Omron Sysmac Studio project 20-1203_20210423 (Sysmac Studio 1.44.0.15, StandardProject)

# Controller new_Controller_0: NX1P2-1140DT version 1.42
Units and slaves: 節點1 : ASDA-A2-E CoE Drive (E001); 節點2 : ASDA-A2-E CoE Drive (E002); 節點3 : ASDA-A2-E CoE Drive (E003); 節點4 : ASDA-A2-E CoE Drive (E004)
Axis MC_AxisLSt5, settings changed from default: AxisType=ServoType, UnitsConversion=EnumElement5, UnitsNumerator=1280000, UnitsDenominator=120, TravelDistancePerWorkRotation=360, WorkGearRatio=3, MaxVelocity=18000, MaxJogVelocity=1800, InPositionCheckTime=500, ZeroPositionBand=0.05
Axis MC_AxisRSt5, settings changed from default: AxisNumber=1, AxisType=ServoType, UnitsConversion=EnumElement5, UnitsNumerator=1280000, UnitsDenominator=120, TravelDistancePerWorkRotation=360, WorkGearRatio=3, MaxVelocity=18000, MaxJogVelocity=1800, InPositionCheckTime=500, ZeroPositionBand=0.05
Axis MC_AxisLSt6, settings changed from default: AxisNumber=2, AxisType=ServoType, UnitsConversion=EnumElement5, UnitsNumerator=1280000, UnitsDenominator=120, TravelDistancePerWorkRotation=360, WorkGearRatio=3, MaxVelocity=18000, MaxJogVelocity=1800, InPositionCheckTime=500, ZeroPositionBand=0.05
Axis MC_AxisRSt6, settings changed from default: AxisNumber=3, AxisType=ServoType, UnitsConversion=EnumElement5, UnitsNumerator=1280000, UnitsDenominator=120, TravelDistancePerWorkRotation=360, WorkGearRatio=3, MaxVelocity=18000, MaxJogVelocity=1800, InPositionCheckTime=500, ZeroPositionBand=0.05
Task PrimaryTask (priority 4, period or condition 4000): prAxisDefineSt5L, prAxisDefineSt5R, prAxisDefineSt6L, prAxisDefineSt6R, prInitial, prIndex, prBowlFeeder, prError, prStation2, prStation3, prStation7, prStation8, prStart, prFeedScrewS5, prCommProgram, prFeedScrewS6, prCycleTime, prBZAndLight, prStation5, prStation6

TYPE StationRecord : STRUCT
    FinishFlag : ARRAY[0..19] OF BOOL;
    OKFlag_1 : ARRAY[0..19] OF BOOL;
    OKFlag_2 : ARRAY[0..19] OF BOOL;
    OKFlag_3 : ARRAY[0..19] OF BOOL;
    OKFlag_4 : ARRAY[0..19] OF BOOL;
    NGFlag_1 : ARRAY[0..19] OF BOOL;
    NGFlag_2 : ARRAY[0..19] OF BOOL;
    NGFlag_3 : ARRAY[0..19] OF BOOL;
    NGFlag_4 : ARRAY[0..19] OF BOOL;
    ErrorRecordData : ARRAY[0..19] OF INT;
END_STRUCT END_TYPE

VAR_GLOBAL CONSTANT
    MC_AxisLSt5 : _sAXIS_REF;  (* at MC://_MC_AX[0] *)
    MC_AxisRSt5 : _sAXIS_REF;  (* at MC://_MC_AX[1] *)
    MC_AxisLSt6 : _sAXIS_REF;  (* at MC://_MC_AX[2] *)
    MC_AxisRSt6 : _sAXIS_REF;  (* at MC://_MC_AX[3] *)
END_VAR
VAR_GLOBAL
    PB_Start1 : BOOL;  (* in_input; at BuiltInIO://cpu/#0/Input_Bit_00; published *)
    PB_Reset1 : BOOL;  (* in_input; at BuiltInIO://cpu/#0/Input_Bit_01; published *)
    PB_Estop1 : BOOL;  (* in_input; at BuiltInIO://cpu/#0/Input_Bit_02; published *)
    PB_Start2 : BOOL;  (* in_input; at BuiltInIO://cpu/#0/Input_Bit_03; published *)
    PB_Reset2 : BOOL;  (* in_input; at BuiltInIO://cpu/#0/Input_Bit_04; published *)
    PB_Estop2 : BOOL;  (* in_input; at BuiltInIO://cpu/#0/Input_Bit_05; published *)
    SNR_AirSource : BOOL;  (* in_input; at BuiltInIO://cpu/#0/Input_Bit_06; published *)
    SNR_Index : BOOL;  (* in_input; at BuiltInIO://cpu/#0/Input_Bit_07; published *)
    LS_S2_THBack1 : BOOL;  (* in_input; at BuiltInIO://cpu/#0/Input_Bit_08; published *)
    LS_S2_THOut1 : BOOL;  (* in_input; at BuiltInIO://cpu/#0/Input_Bit_09; published *)
    LS_S2_THBack2 : BOOL;  (* in_input; at BuiltInIO://cpu/#0/Input_Bit_10; published *)
    LS_S2_THOut2 : BOOL;  (* in_input; at BuiltInIO://cpu/#0/Input_Bit_11; published *)
    LS_S2_MoveBack : BOOL;  (* in_input; at BuiltInIO://cpu/#0/Input_Bit_12; published *)
    LS_S2_MoveOut : BOOL;  (* in_input; at BuiltInIO://cpu/#0/Input_Bit_13; published *)
    SNR_S2_Feed : BOOL;  (* in_input; at BuiltInIO://cpu/#0/Input_Bit_14; published *)
    SNR_S2_Full : BOOL;  (* in_input; at BuiltInIO://cpu/#0/Input_Bit_15; published *)
    LS_S3_THBack1 : BOOL;  (* in_input; at BuiltInIO://cpu/#0/Input_Bit_16; published *)
    LS_S3_THOut1 : BOOL;  (* in_input; at BuiltInIO://cpu/#0/Input_Bit_17; published *)
    LS_S3_THBack2 : BOOL;  (* in_input; at BuiltInIO://cpu/#0/Input_Bit_18; published *)
    LS_S3_THOut2 : BOOL;  (* in_input; at BuiltInIO://cpu/#0/Input_Bit_19; published *)
    LS_S3_MoveBack : BOOL;  (* in_input; at BuiltInIO://cpu/#0/Input_Bit_20; published *)
    LS_S3_MoveOut : BOOL;  (* in_input; at BuiltInIO://cpu/#0/Input_Bit_21; published *)
    SNR_S3_Feed : BOOL;  (* in_input; at BuiltInIO://cpu/#0/Input_Bit_22; published *)
    SNR_S3_Full : BOOL;  (* in_input; at BuiltInIO://cpu/#0/Input_Bit_23; published *)
    LS_S5_UpDownBack : BOOL;  (* in_input; at IOBus://unit#2/Input Bit 16 bits/Input Bit 00; published *)
    LS_S5_UpDownOut : BOOL;  (* in_input; at IOBus://unit#2/Input Bit 16 bits/Input Bit 01; published *)
    LS_S5_FixBack : BOOL;  (* in_input; at IOBus://unit#2/Input Bit 16 bits/Input Bit 02; published *)
    LS_S5_FixOut : BOOL;  (* in_input; at IOBus://unit#2/Input Bit 16 bits/Input Bit 03; published *)
    SNR_S5_L_Check : BOOL;  (* in_input; at IOBus://unit#2/Input Bit 16 bits/Input Bit 04; published *)
    SNR_S5_R_Check : BOOL;  (* in_input; at IOBus://unit#2/Input Bit 16 bits/Input Bit 05; published *)
    SNR_S5_L_Feed : BOOL;  (* in_input; at IOBus://unit#2/Input Bit 16 bits/Input Bit 06; published *)
    SNR_S5_R_Feed : BOOL;  (* in_input; at IOBus://unit#2/Input Bit 16 bits/Input Bit 07; published *)
    LS_S6_UpDownBack : BOOL;  (* in_input; at IOBus://unit#2/Input Bit 16 bits/Input Bit 08; published *)
    LS_S6_UpDownOut : BOOL;  (* in_input; at IOBus://unit#2/Input Bit 16 bits/Input Bit 09; published *)
    LS_S6_FixBack : BOOL;  (* in_input; at IOBus://unit#2/Input Bit 16 bits/Input Bit 10; published *)
    LS_S6_FixOut : BOOL;  (* in_input; at IOBus://unit#2/Input Bit 16 bits/Input Bit 11; published *)
    SNR_S6_L_Check : BOOL;  (* in_input; at IOBus://unit#2/Input Bit 16 bits/Input Bit 12; published *)
    SNR_S6_R_Check : BOOL;  (* in_input; at IOBus://unit#2/Input Bit 16 bits/Input Bit 13; published *)
    SNR_S6_L_Feed : BOOL;  (* in_input; at IOBus://unit#2/Input Bit 16 bits/Input Bit 14; published *)
    SNR_S6_R_Feed : BOOL;  (* in_input; at IOBus://unit#2/Input Bit 16 bits/Input Bit 15; published *)
    SNR_S5_Full : BOOL;  (* in_input; at IOBus://unit#3/Input Bit 16 bits/Input Bit 00; published *)
    SNR_S6_Full : BOOL;  (* in_input; at IOBus://unit#3/Input Bit 16 bits/Input Bit 01; published *)
    LS_S7_MoveBack1 : BOOL;  (* in_input; at IOBus://unit#3/Input Bit 16 bits/Input Bit 02; published *)
    LS_S7_MoveOut1 : BOOL;  (* in_input; at IOBus://unit#3/Input Bit 16 bits/Input Bit 03; published *)
    LS_S7_MoveBack2 : BOOL;  (* in_input; at IOBus://unit#3/Input Bit 16 bits/Input Bit 04; published *)
    LS_S7_MoveOut2 : BOOL;  (* in_input; at IOBus://unit#3/Input Bit 16 bits/Input Bit 05; published *)
    LS_S7_MoveBack3 : BOOL;  (* in_input; at IOBus://unit#3/Input Bit 16 bits/Input Bit 06; published *)
    LS_S7_MoveOut3 : BOOL;  (* in_input; at IOBus://unit#3/Input Bit 16 bits/Input Bit 07; published *)
    LS_S7_MoveBack4 : BOOL;  (* in_input; at IOBus://unit#3/Input Bit 16 bits/Input Bit 08; published *)
    LS_S7_MoveOut4 : BOOL;  (* in_input; at IOBus://unit#3/Input Bit 16 bits/Input Bit 09; published *)
    SNR_S7_Full : BOOL;  (* in_input; at IOBus://unit#3/Input Bit 16 bits/Input Bit 10; published *)
    LS_S8_MoveBack : BOOL;  (* in_input; at IOBus://unit#3/Input Bit 16 bits/Input Bit 11; published *)
    LS_S8_MoveOut : BOOL;  (* in_input; at IOBus://unit#3/Input Bit 16 bits/Input Bit 12; published *)
    LS_S5_IndexFixBack : BOOL;  (* in_input; at IOBus://unit#3/Input Bit 16 bits/Input Bit 13; published *)
    LS_S5_IndexFixOut : BOOL;  (* in_input; at IOBus://unit#3/Input Bit 16 bits/Input Bit 14; published *)
    LS_S6_IndexFixBack : BOOL;  (* in_input; at IOBus://unit#3/Input Bit 16 bits/Input Bit 15; published *)
    LS_S6_IndexFixOut : BOOL;  (* in_input; at IOBus://unit#4/Input Bit 16 bits/Input Bit 00; published *)
    RY_Index : BOOL;  (* output; at BuiltInIO://cpu/#0/Output_Bit_00; published *)
    RY_S2_Full : BOOL;  (* output; at BuiltInIO://cpu/#0/Output_Bit_01; published *)
    RY_S2_Feed : BOOL;  (* output; at BuiltInIO://cpu/#0/Output_Bit_02; published *)
    RY_S3_Full : BOOL;  (* output; at BuiltInIO://cpu/#0/Output_Bit_03; published *)
    RY_S3_Feed : BOOL;  (* output; at BuiltInIO://cpu/#0/Output_Bit_04; published *)
    RY_S5_Full : BOOL;  (* output; at BuiltInIO://cpu/#0/Output_Bit_05; published *)
    RY_S5_Feed : BOOL;  (* output; at BuiltInIO://cpu/#0/Output_Bit_06; published *)
    RY_S6_Full : BOOL;  (* output; at BuiltInIO://cpu/#0/Output_Bit_07; published *)
    RY_S6_Feed : BOOL;  (* output; at BuiltInIO://cpu/#0/Output_Bit_08; published *)
    SOL_S2_THBack1 : BOOL;  (* output; at BuiltInIO://cpu/#0/Output_Bit_09; published *)
    SOL_S2_THOut1 : BOOL;  (* output; at BuiltInIO://cpu/#0/Output_Bit_10; published *)
    SOL_S2_THBack2 : BOOL;  (* output; at BuiltInIO://cpu/#0/Output_Bit_11; published *)
    SOL_S2_THOut2 : BOOL;  (* output; at BuiltInIO://cpu/#0/Output_Bit_12; published *)
    SOL_S2_Move : BOOL;  (* output; at BuiltInIO://cpu/#0/Output_Bit_13; published *)
    SOL_S3_THBack1 : BOOL;  (* output; at BuiltInIO://cpu/#0/Output_Bit_14; published *)
    SOL_S3_THOut1 : BOOL;  (* output; at BuiltInIO://cpu/#0/Output_Bit_15; published *)
    SOL_S3_THBack2 : BOOL;  (* output; at IOBus://unit#5/Output Bit 16 bits/Output Bit 00; published *)
    SOL_S3_THOut2 : BOOL;  (* output; at IOBus://unit#5/Output Bit 16 bits/Output Bit 01; published *)
    SOL_S3_Move : BOOL;  (* output; at IOBus://unit#5/Output Bit 16 bits/Output Bit 02; published *)
    SOL_S5_Feed : BOOL;  (* output; at IOBus://unit#5/Output Bit 16 bits/Output Bit 03; published *)
    SOL_S5_UpDown : BOOL;  (* output; at IOBus://unit#5/Output Bit 16 bits/Output Bit 04; published *)
    SOL_S5_Clamp : BOOL;  (* output; at IOBus://unit#5/Output Bit 16 bits/Output Bit 05; published *)
    SOL_S5_Fix : BOOL;  (* output; at IOBus://unit#5/Output Bit 16 bits/Output Bit 06; published *)
    SOL_S6_Feed : BOOL;  (* output; at IOBus://unit#5/Output Bit 16 bits/Output Bit 07; published *)
    SOL_S6_UpDown : BOOL;  (* output; at IOBus://unit#5/Output Bit 16 bits/Output Bit 08; published *)
    SOL_S6_Clamp : BOOL;  (* output; at IOBus://unit#5/Output Bit 16 bits/Output Bit 09; published *)
    SOL_S6_Fix : BOOL;  (* output; at IOBus://unit#5/Output Bit 16 bits/Output Bit 10; published *)
    SOL_S7_Move1 : BOOL;  (* output; at IOBus://unit#5/Output Bit 16 bits/Output Bit 11; published *)
    SOL_S7_Move2 : BOOL;  (* output; at IOBus://unit#5/Output Bit 16 bits/Output Bit 12; published *)
    SOL_S7_Move3 : BOOL;  (* output; at IOBus://unit#5/Output Bit 16 bits/Output Bit 13; published *)
    SOL_S7_Move4 : BOOL;  (* output; at IOBus://unit#5/Output Bit 16 bits/Output Bit 14; published *)
    SOL_S8_Move : BOOL;  (* output; at IOBus://unit#5/Output Bit 16 bits/Output Bit 15; published *)
    SOL_S5_IndexFixBack : BOOL;  (* output; at IOBus://unit#6/Output Bit 16 bits/Output Bit 00; published *)
    SOL_S5_IndexFixOut : BOOL;  (* output; at IOBus://unit#6/Output Bit 16 bits/Output Bit 01; published *)
    SOL_S6_IndexFixBack : BOOL;  (* output; at IOBus://unit#6/Output Bit 16 bits/Output Bit 02; published *)
    SOL_S6_IndexFixOut : BOOL;  (* output; at IOBus://unit#6/Output Bit 16 bits/Output Bit 03; published *)
    BZ : BOOL;  (* output; at IOBus://unit#6/Output Bit 16 bits/Output Bit 04; published *)
    YL : BOOL;  (* output; at IOBus://unit#6/Output Bit 16 bits/Output Bit 05; published *)
    GL : BOOL;  (* output; at IOBus://unit#6/Output Bit 16 bits/Output Bit 06; published *)
    RL : BOOL;  (* output; at IOBus://unit#6/Output Bit 16 bits/Output Bit 07; published *)
    SOL_S2_Fix : BOOL;  (* output; at IOBus://unit#6/Output Bit 16 bits/Output Bit 08; published *)
    SOL_S3_Fix : BOOL;  (* output; at IOBus://unit#6/Output Bit 16 bits/Output Bit 09; published *)
END_VAR
VAR_GLOBAL RETAIN
    HMI_FeedScrewTime : ARRAY[0..1] OF INT;  (* published *)
END_VAR
VAR_GLOBAL
    HMIPB_RY_Index : BOOL;  (* HMIPB; published *)
    HMIPB_SOL_S2_THBack1 : BOOL;  (* HMIPB; published *)
    HMIPB_SOL_S2_THOut1 : BOOL;  (* HMIPB; published *)
    HMIPB_SOL_S2_THBack2 : BOOL;  (* HMIPB; published *)
    HMIPB_SOL_S2_THOut2 : BOOL;  (* HMIPB; published *)
    HMIPB_SOL_S2_Move : BOOL;  (* HMIPB; published *)
    HMIPB_SOL_S3_THBack1 : BOOL;  (* HMIPB; published *)
    HMIPB_SOL_S3_THOut1 : BOOL;  (* HMIPB; published *)
    HMIPB_SOL_S3_THBack2 : BOOL;  (* HMIPB; published *)
    HMIPB_SOL_S3_THOut2 : BOOL;  (* HMIPB; published *)
    HMIPB_SOL_S3_Move : BOOL;  (* HMIPB; published *)
    HMIPB_SOL_S5_Feed : BOOL;  (* HMIPB; published *)
    HMIPB_SOL_S5_UpDown : BOOL;  (* HMIPB; published *)
    HMIPB_SOL_S5_Clamp : BOOL;  (* HMIPB; published *)
    HMIPB_SOL_S5_Fix : BOOL;  (* HMIPB; published *)
    HMIPB_SOL_S6_Feed : BOOL;  (* HMIPB; published *)
    HMIPB_SOL_S6_UpDown : BOOL;  (* HMIPB; published *)
    HMIPB_SOL_S6_Clamp : BOOL;  (* HMIPB; published *)
    HMIPB_SOL_S6_Fix : BOOL;  (* HMIPB; published *)
    HMIPB_SOL_S7_Move1 : BOOL;  (* HMIPB; published *)
    HMIPB_SOL_S7_Move2 : BOOL;  (* HMIPB; published *)
    HMIPB_SOL_S7_Move3 : BOOL;  (* HMIPB; published *)
    HMIPB_SOL_S7_Move4 : BOOL;  (* HMIPB; published *)
    HMIPB_SOL_S8_Move : BOOL;  (* HMIPB; published *)
    HMIPB_SOL_IndexFixBack : BOOL;  (* HMIPB; published *)
    HMIPB_SOL_IndexFixOut : BOOL;  (* HMIPB; published *)
    HMIPB_SOL_S2_Fix : BOOL;  (* HMIPB; published *)
    HMIPB_SOL_S3_Fix : BOOL;  (* HMIPB; published *)
    HMIPB_S2Feed : BOOL;  (* published *)
    HMIPB_S3Feed : BOOL;  (* published *)
    HMIPB_S5Feed : BOOL;  (* published *)
    HMIPB_S6Feed : BOOL;  (* published *)
    HMIPB_DisableS2 : BOOL;  (* published *)
    HMIPB_DisableS3 : BOOL;  (* published *)
    BackoutStart : ARRAY[0..3] OF BOOL;
    BackoutBusy : ARRAY[0..3] OF BOOL;
    ScrewStartS5LFW : BOOL;
    ScrewStartS5LRW : BOOL;
    ScrewStartS5RFW : BOOL;
    ScrewStartS5RRW : BOOL;
    ScrewStartS6LFW : BOOL;
    ScrewStartS6LRW : BOOL;
    ScrewStartS6RFW : BOOL;
    ScrewStartS6RRW : BOOL;
    Error_PB_Estop1 : BOOL;  (* Error; published *)
    Error_PB_Estop2 : BOOL;  (* Error; published *)
    Error_SNR_AirSource : BOOL;  (* Error; published *)
    Error_SNR_Index : BOOL;  (* Error; published *)
    Error_LS_S2_THBack1 : BOOL;  (* Error; published *)
    Error_LS_S2_THOut1 : BOOL;  (* Error; published *)
    Error_LS_S2_THBack2 : BOOL;  (* Error; published *)
    Error_LS_S2_THOut2 : BOOL;  (* Error; published *)
    Error_LS_S2_MoveBack : BOOL;  (* Error; published *)
    Error_LS_S2_MoveOut : BOOL;  (* Error; published *)
    Error_SNR_S2_Feed : BOOL;  (* Error; published *)
    Error_SNR_S2_Full : BOOL;  (* Error; published *)
    Error_LS_S3_THBack1 : BOOL;  (* Error; published *)
    Error_LS_S3_THOut1 : BOOL;  (* Error; published *)
    Error_LS_S3_THBack2 : BOOL;  (* Error; published *)
    Error_LS_S3_THOut2 : BOOL;  (* Error; published *)
    Error_LS_S3_MoveBack : BOOL;  (* Error; published *)
    Error_LS_S3_MoveOut : BOOL;  (* Error; published *)
    Error_SNR_S3_Feed : BOOL;  (* Error; published *)
    Error_SNR_S3_Full : BOOL;  (* Error; published *)
    Error_LS_S5_UpDownBack : BOOL;  (* Error; published *)
    Error_LS_S5_UpDownOut : BOOL;  (* Error; published *)
    Error_LS_S5_FixBack : BOOL;  (* Error; published *)
    Error_LS_S5_FixOut : BOOL;  (* Error; published *)
    Error_SNR_S5_L_Check : BOOL;  (* Error; published *)
    Error_SNR_S5_R_Check : BOOL;  (* Error; published *)
    Error_SNR_S5_L_Feed : BOOL;  (* Error; published *)
    Error_SNR_S5_R_Feed : BOOL;  (* Error; published *)
    Error_LS_S6_UpDownBack : BOOL;  (* Error; published *)
    Error_LS_S6_UpDownOut : BOOL;  (* Error; published *)
    Error_LS_S6_FixBack : BOOL;  (* Error; published *)
    Error_LS_S6_FixOut : BOOL;  (* Error; published *)
    Error_SNR_S6_L_Check : BOOL;  (* Error; published *)
    Error_SNR_S6_R_Check : BOOL;  (* Error; published *)
    Error_SNR_S6_L_Feed : BOOL;  (* Error; published *)
    Error_SNR_S6_R_Feed : BOOL;  (* Error; published *)
    Error_SNR_S5_Full : BOOL;  (* Error; published *)
    Error_SNR_S6_Full : BOOL;  (* Error; published *)
    Error_LS_S7_MoveBack1 : BOOL;  (* Error; published *)
    Error_LS_S7_MoveOut1 : BOOL;  (* Error; published *)
    Error_LS_S7_MoveBack2 : BOOL;  (* Error; published *)
    Error_LS_S7_MoveOut2 : BOOL;  (* Error; published *)
    Error_LS_S7_MoveBack3 : BOOL;  (* Error; published *)
    Error_LS_S7_MoveOut3 : BOOL;  (* Error; published *)
    Error_LS_S7_MoveBack4 : BOOL;  (* Error; published *)
    Error_LS_S7_MoveOut4 : BOOL;  (* Error; published *)
    Error_SNR_S7_Full : BOOL;  (* Error; published *)
    Error_LS_S8_MoveBack : BOOL;  (* Error; published *)
    Error_LS_S8_MoveOut : BOOL;  (* Error; published *)
    Error_LS_S5_IndexFixBack : BOOL;  (* Error; published *)
    Error_LS_S5_IndexFixOut : BOOL;  (* Error; published *)
    Error_LS_S6_IndexFixBack : BOOL;  (* Error; published *)
    Error_LS_S6_IndexFixOut : BOOL;  (* Error; published *)
    AutoStatus : bool;  (* status; published *)
    MachineRunStatus : bool;  (* published *)
    SystemReadyStatus : bool;  (* published *)
    Manual2AutoFlag : bool;  (* status; published *)
    IndexCanRunStatus : bool;  (* status; published *)
    FeedStartFlag : ARRAY[0..1] OF bool;  (* status; published *)
    FeedFlowS2 : INT;  (* status *)
    FeedFlowS3 : INT;
    ScrewStartFlag : ARRAY[0..3] OF bool;
    ErrorStatus_MachineStop : bool;  (* status; published *)
    ErrorStatus_MachineNonStop : bool;  (* status; published *)
    ErrorStatus_MachineStop_Record : bool;  (* status; published *)
END_VAR
VAR_GLOBAL RETAIN
    OBJScrewInTube : ARRAY[0..3] OF INT;  (* status; published *)
    OBJScrewInClip : ARRAY[0..3] OF INT;  (* status; published *)
END_VAR
VAR_GLOBAL
    HMIPB_AlarmResetAxisLSt5 : BOOL;  (* published *)
    HMIPB_AlarmResetAxisRSt5 : BOOL;  (* published *)
    HMIPB_AlarmResetAxisLSt6 : BOOL;  (* published *)
    HMIPB_AlarmResetAxisRSt6 : BOOL;  (* published *)
    HMIPB_ServoStopAxisLSt5 : BOOL;  (* published *)
    HMIPB_ServoStopAxisRSt5 : BOOL;  (* published *)
    HMIPB_ServoStopAxisLSt6 : BOOL;  (* published *)
    HMIPB_ServoStopAxisRSt6 : BOOL;  (* published *)
    HMIPB_FW_AxisLSt5 : BOOL;  (* published *)
    HMIPB_RW_AxisLSt5 : BOOL;  (* published *)
    HMIPB_FW_AxisRSt5 : BOOL;  (* published *)
    HMIPB_RW_AxisRSt5 : BOOL;  (* published *)
    HMIPB_FW_AxisLSt6 : BOOL;  (* published *)
    HMIPB_RW_AxisLSt6 : BOOL;  (* published *)
    HMIPB_FW_AxisRSt6 : BOOL;  (* published *)
    HMIPB_RW_AxisRSt6 : BOOL;  (* published *)
END_VAR
VAR_GLOBAL RETAIN
    HMIPB_ServoON_AxisLSt5 : BOOL;  (* published *)
    HMIPB_ServoON_AxisRSt5 : BOOL;  (* published *)
    HMIPB_ServoON_AxisLSt6 : BOOL;  (* published *)
    HMIPB_ServoON_AxisRSt6 : BOOL;  (* published *)
END_VAR
VAR_GLOBAL
    HMIPB_SerchHome_AxisLSt5 : BOOL;  (* published *)
    HMIPB_SerchHome_AxisRSt5 : BOOL;  (* published *)
    HMIPB_SerchHome_AxisLSt6 : BOOL;  (* published *)
    HMIPB_SerchHome_AxisRSt6 : BOOL;  (* published *)
    OutPutFeedRYS5 : BOOL;
    OutPutFeedRYS6 : BOOL;
    Flash1s : BOOL;
    HMIPB_ResetCount : BOOL;
    ResetAddress : ARRAY[0..3] OF bool;
    HMI_AllCount : UDINT;
END_VAR
VAR_GLOBAL RETAIN
    HMI_FeededS2 : BOOL;  (* published *)
    HMI_FeededS3 : BOOL;  (* published *)
    HMI_ScrewTorque_St5_L : LREAL;  (* published *)
    HMI_ScrewSpeed_St5_L : LREAL;  (* published *)
    HMI_ScrewTorque_St5_R : LREAL;  (* published *)
    HMI_ScrewSpeed_St5_R : LREAL;  (* published *)
    HMI_ScrewTorque_St6_L : LREAL;  (* published *)
    HMI_ScrewSpeed_St6_L : LREAL;  (* published *)
    HMI_ScrewTorque_St6_R : LREAL;  (* published *)
    HMI_ScrewSpeed_St6_R : LREAL;  (* published *)
    HMI_BackOutTorque_St5_R : LREAL;  (* published *)
    HMI_BackOutTorque_St5_L : LREAL;  (* published *)
    HMI_BackOutTorque_St6_R : LREAL;  (* published *)
    HMI_BackOutTorque_St6_L : LREAL;  (* published *)
    HMI_BackOutAngle_St5_R : LREAL;  (* published *)
    HMI_BackOutAngle_St5_L : LREAL;  (* published *)
    HMI_BackOutAngle_St6_L : LREAL;  (* published *)
    HMI_BackOutAngle_St6_R : LREAL;  (* published *)
    HMI_LimitAngle_St5_L : LREAL;  (* published *)
    HMI_LimitAngle_St5_R : LREAL;  (* published *)
    HMI_LimitAngle_St6_L : LREAL;  (* published *)
    HMI_LimitAngle_St6_R : LREAL;  (* published *)
    HMI_NoScrewAngle_St5_L : LREAL;  (* published *)
    HMI_NoScrewAngle_St5_R : LREAL;  (* published *)
    HMI_NoScrewAngle_St6_L : LREAL;  (* published *)
    HMI_NoScrewAngle_St6_R : LREAL;  (* published *)
    HMI_Find_St5_L : LINT;  (* published *)
    HMI_Find_St5_R : LINT;  (* published *)
    HMI_Find_St6_L : LINT;  (* published *)
    HMI_Find_St6_R : LINT;  (* published *)
    OKCount : UDINT;  (* published *)
    TotalCount : UDINT;  (* published *)
END_VAR
VAR_GLOBAL
    HMI_CycleTime : LINT;  (* published *)
    HMIShow_Homed : ARRAY[0..3] OF BOOL;  (* published *)
    HMIShow_Error : ARRAY[0..3] OF BOOL;  (* published *)
    HMIShow_POT : ARRAY[0..3] OF BOOL;  (* published *)
    HMIShow_NOT : ARRAY[0..3] OF BOOL;  (* published *)
    HMIShow_CurrentPosition : ARRAY[0..3] OF LREAL;  (* published *)
    HMIShow_CurrentSpeed : ARRAY[0..3] OF LREAL;  (* published *)
    HMIShow_CurrentTorque : ARRAY[0..3] OF LREAL;  (* published *)
    HMIShow_OK2 : ARRAY[0..3] OF Bool;  (* published *)
    HMIShow_OK3 : ARRAY[0..3] OF Bool;  (* published *)
    HMIShow_OK4 : ARRAY[0..3] OF Bool;  (* published *)
    HMIShow_OK5 : ARRAY[0..3] OF Bool;  (* published *)
    HMIShow_OK6 : ARRAY[0..3] OF Bool;  (* published *)
    HMIShow_OK7 : ARRAY[0..3] OF Bool;  (* published *)
    HMIShow_OK8 : ARRAY[0..3] OF Bool;  (* published *)
    HMIShow_NG2 : ARRAY[0..3] OF Bool;  (* published *)
    HMIShow_NG3 : ARRAY[0..3] OF Bool;  (* published *)
    HMIShow_NG4 : ARRAY[0..3] OF Bool;  (* published *)
    HMIShow_NG5 : ARRAY[0..3] OF Bool;  (* published *)
    HMIShow_NG6 : ARRAY[0..3] OF Bool;  (* published *)
    HMIShow_NG7 : ARRAY[0..3] OF Bool;  (* published *)
    HMIShow_NG8 : ARRAY[0..3] OF Bool;  (* published *)
END_VAR
VAR_GLOBAL RETAIN
    HMI_ItemNotExistsDelayTime : ARRAY[0..6] OF LINT;  (* published *)
    HMI_ItemExistsDelayTime : ARRAY[0..6] OF LINT;  (* published *)
    HMI_ItemNotExistsErrorTime : ARRAY[0..6] OF LINT;  (* published *)
    IndexData0 : StationRecord;  (* published *)
    IndexData1 : StationRecord;  (* published *)
    IndexData2 : StationRecord;  (* published *)
    IndexData3 : StationRecord;  (* published *)
    IndexData4 : StationRecord;  (* published *)
    IndexData5 : StationRecord;  (* published *)
    IndexData6 : StationRecord;  (* published *)
    IndexData7 : StationRecord;  (* published *)
    IndexData8 : StationRecord;  (* published *)
END_VAR

PROGRAM prFeedScrewS5
VAR
    SolFeed : fbSingleSolRy;
    ErrorState : BOOL;
    AutoFlow : INT;
    TON1 : TON;
    TON2 : TON;
    TON3 : TON;
    Check1 : fbCheckScrew_Tube;
    Check2 : fbCheckScrew_Tube;
    RTRIG1 : R_TRIG;
END_VAR
VAR_EXTERNAL
    AutoStatus : bool;
    SystemReadyStatus : bool;
    HMIPB_SOL_S5_Feed : BOOL;
    SOL_S5_Feed : BOOL;
    FeedStartFlag : ARRAY[0..1] OF bool;
    HMI_FeedScrewTime : ARRAY[0..1] OF INT;
    RY_S5_Feed : BOOL;
    OutPutFeedRYS5 : BOOL;
    LS_S5_UpDownOut : BOOL;
    SNR_S5_L_Feed : BOOL;
    PB_Reset1 : BOOL;
    PB_Reset2 : BOOL;
    Error_SNR_S5_L_Feed : BOOL;
    SNR_S5_R_Feed : BOOL;
    Error_SNR_S5_R_Feed : BOOL;
    OBJScrewInClip : ARRAY[0..3] OF INT;
    OBJScrewInTube : ARRAY[0..3] OF INT;
    LS_S5_UpDownBack : BOOL;
    SOL_S5_UpDown : BOOL;
    HMIPB_S5Feed : BOOL;
END_VAR
//********************************************************************
//Check
//********************************************************************
Check1(
	inClearSingle:=LS_S5_UpDownOut,
	inFeedSNR:=SNR_S5_L_Feed,
	inBlowSOL:=SOL_S5_Feed,
	inReset:=PB_Reset1 OR PB_Reset2,
	outError=>Error_SNR_S5_L_Feed,
	inoutScrewInClip:=OBJScrewInClip[0],
	inoutScrewInTube:=OBJScrewInTube[0]);
Check2(
	inClearSingle:=LS_S5_UpDownOut,
	inFeedSNR:=SNR_S5_R_Feed,
	inBlowSOL:=SOL_S5_Feed,
	inReset:=PB_Reset1 OR PB_Reset2,
	outError=>Error_SNR_S5_R_Feed,
	inoutScrewInClip:=OBJScrewInClip[1],
	inoutScrewInTube:=OBJScrewInTube[1]);
//********************************************************************
//Manual
//********************************************************************
//Feed screw sol
SolFeed(
	inAutoStatus:=AutoStatus,
	inAutoFlowSet:=AutoFlow=3,
	inAutoFlowReset:=AutoFlow=4,
	inInterLockBack:=TRUE,
	inInterLockOut:=NOT(SOL_S5_UpDown) AND LS_S5_UpDownBack,
	outSol=>	SOL_S5_Feed);
//********************************************************************
//Auto
//********************************************************************
IF LS_S5_UpDownOut AND SOL_S5_UpDown THEN
	FeedStartFlag[0]:=TRUE;
END_IF;
ErrorState:=FALSE;
//power on=0
IF NOT(SystemReadyStatus) OR ErrorState THEN
	AutoFlow:=0;
	FeedStartFlag[0]:=FALSE;
END_IF;
//idle=1
IF AutoFlow=0 AND NOT(NOT(SystemReadyStatus) OR ErrorState) THEN
	AutoFlow:=1;
END_IF;
IF AutoFlow=6 AND NOT(OutPutFeedRYS5) THEN
	AutoFlow:=1;
END_IF;
//Feed RY on=2
RTRIG1(Clk:=HMIPB_SOL_S5_Feed);
IF AutoFlow=1 AND ((FeedStartFlag[0] AND AutoStatus) OR (RTRIG1.Q AND NOT(AutoStatus))) THEN
	AutoFlow:=2;
	OutPutFeedRYS5:=TRUE;
END_IF;
//Feed Sol on=3
TON1(In:=AutoFlow=2 AND RY_S5_Feed, PT:=t#800ms);
//
IF AutoFlow=2 AND TON1.Q THEN
	AutoFlow:=3;
END_IF;
IF AutoFlow=5 AND NOT(TON3.Q) AND FeedStartFlag[0] THEN
	AutoFlow:=3;
END_IF;
//Feed Sol off=4
TON2(In:=AutoFlow=3 AND SOL_S5_Feed, PT:=NanoSecToTime(HMI_FeedScrewTime[0]*100000000));
IF AutoFlow=3 AND ((TON2.Q AND AutoStatus) OR RTRIG1.Q AND NOT(AutoStatus)) THEN
	AutoFlow:=4;
END_IF;
//Feed Finish=5
IF AutoFlow=4 AND NOT(SOL_S5_Feed) THEN
	AutoFlow:=5;
	FeedStartFlag[0]:=FALSE;
END_IF;
//Feed RY off=6
TON3(In:=AutoFlow=5, PT:=t#5s);
IF AutoFlow=5 AND TON3.Q THEN
	AutoFlow:=6;
	OutPutFeedRYS5:=FALSE;
END_IF;
END_PROGRAM

PROGRAM prFeedScrewS6
VAR
    SolFeed : fbSingleSolRy;
    ErrorState : BOOL;
    AutoFlow : INT;
    TON1 : TON;
    TON2 : TON;
    TON3 : TON;
    Check1 : fbCheckScrew_Tube;
    Check2 : fbCheckScrew_Tube;
    RTRIG1 : R_TRIG;
END_VAR
VAR_EXTERNAL
    AutoStatus : bool;
    SystemReadyStatus : bool;
    HMIPB_SOL_S5_Feed : BOOL;
    SOL_S5_Feed : BOOL;
    FeedStartFlag : ARRAY[0..1] OF bool;
    HMI_FeedScrewTime : ARRAY[0..1] OF INT;
    RY_S5_Feed : BOOL;
    OutPutFeedRYS5 : BOOL;
    LS_S5_UpDownOut : BOOL;
    SNR_S5_L_Feed : BOOL;
    PB_Reset1 : BOOL;
    PB_Reset2 : BOOL;
    Error_SNR_S5_L_Feed : BOOL;
    SNR_S5_R_Feed : BOOL;
    Error_SNR_S5_R_Feed : BOOL;
    LS_S6_UpDownOut : BOOL;
    SNR_S6_L_Feed : BOOL;
    SOL_S6_Feed : BOOL;
    Error_SNR_S6_L_Feed : BOOL;
    SNR_S6_R_Feed : BOOL;
    Error_SNR_S6_R_Feed : BOOL;
    HMIPB_SOL_S6_Feed : BOOL;
    RY_S6_Feed : BOOL;
    OutPutFeedRYS6 : BOOL;
    OBJScrewInClip : ARRAY[0..3] OF INT;
    OBJScrewInTube : ARRAY[0..3] OF INT;
    LS_S6_UpDownBack : BOOL;
    SOL_S2_Fix : BOOL;
    SOL_S6_UpDown : BOOL;
END_VAR
//********************************************************************
//Check
//********************************************************************
Check1(
	inClearSingle:=LS_S6_UpDownOut,
	inFeedSNR:=SNR_S6_L_Feed,
	inBlowSOL:=SOL_S6_Feed,
	inReset:=PB_Reset1 OR PB_Reset2,
	outError=>Error_SNR_S6_L_Feed,
	inoutScrewInClip:=OBJScrewInClip[2],
	inoutScrewInTube:=OBJScrewInTube[2]);
Check2(
	inClearSingle:=LS_S6_UpDownOut,
	inFeedSNR:=SNR_S6_R_Feed,
	inBlowSOL:=SOL_S6_Feed,
	inReset:=PB_Reset1 OR PB_Reset2,
	outError=>Error_SNR_S6_R_Feed,
	inoutScrewInClip:=OBJScrewInClip[3],
	inoutScrewInTube:=OBJScrewInTube[3]);
//********************************************************************
//Manual
//********************************************************************
//Feed screw sol
SolFeed(
	inAutoStatus:=AutoStatus,
	inAutoFlowSet:=AutoFlow=3,
	inAutoFlowReset:=AutoFlow=4,
	inInterLockBack:=TRUE,
	inInterLockOut:=NOT(SOL_S6_UpDown) AND LS_S6_UpDownBack,
	outSol=>	SOL_S6_Feed);
//********************************************************************
//Auto
//********************************************************************
IF LS_S6_UpDownOut AND SOL_S6_UpDown THEN
	FeedStartFlag[1]:=TRUE;
END_IF;
ErrorState:=FALSE;
//power on=0
IF NOT(SystemReadyStatus) OR ErrorState THEN
	AutoFlow:=0;
	FeedStartFlag[1]:=FALSE;
END_IF;
//idle=1
IF AutoFlow=0 AND NOT(NOT(SystemReadyStatus) OR ErrorState) THEN
	AutoFlow:=1;
END_IF;
IF AutoFlow=6 AND NOT(OutPutFeedRYS6) THEN
	AutoFlow:=1;
END_IF;
//Feed RY on=2
RTRIG1(Clk:=HMIPB_SOL_S6_Feed);
IF AutoFlow=1 AND ((FeedStartFlag[1] AND AutoStatus) OR (RTRIG1.Q AND NOT(AutoStatus))) THEN
	AutoFlow:=2;
	OutPutFeedRYS6:=TRUE;
END_IF;
//Feed Sol on=3
TON1(In:=AutoFlow=2 AND RY_S6_Feed, PT:=t#800ms);
//
IF AutoFlow=2 AND TON1.Q THEN
	AutoFlow:=3;
END_IF;
IF AutoFlow=5 AND NOT(TON3.Q) AND FeedStartFlag[1] THEN
	AutoFlow:=3;
END_IF;
//Feed Sol off=4
TON2(In:=AutoFlow=3 AND SOL_S6_Feed, PT:=NanoSecToTime(HMI_FeedScrewTime[1]*100000000));
IF AutoFlow=3 AND ((TON2.Q AND AutoStatus) OR RTRIG1.Q AND NOT(AutoStatus)) THEN
	AutoFlow:=4;
END_IF;
//Feed Finish=5
IF AutoFlow=4 AND NOT(SOL_S6_Feed) THEN
	AutoFlow:=5;
	FeedStartFlag[1]:=FALSE;
END_IF;
//Feed RY off=6
TON3(In:=AutoFlow=5, PT:=t#5s);
IF AutoFlow=5 AND TON3.Q THEN
	AutoFlow:=6;
	OutPutFeedRYS6:=FALSE;
END_IF;
END_PROGRAM

PROGRAM prIndex
VAR
    SOLIndexFixS5 : fbDoubleSolRy;
    SOLIndexFixS6 : fbDoubleSolRy;
    AutoFlow : INT;
    ErrorStatus : BOOL;
    R_TRIG_1 : R_TRIG;
    AllStationFinish : BOOL;
END_VAR
VAR_EXTERNAL
    LS_S2_MoveBack : BOOL;
    SOL_S2_Move : BOOL;
    LS_S3_MoveBack : BOOL;
    SOL_S3_Move : BOOL;
    LS_S5_UpDownBack : BOOL;
    SOL_S5_UpDown : BOOL;
    LS_S6_UpDownBack : BOOL;
    SOL_S6_UpDown : BOOL;
    LS_S7_MoveBack1 : BOOL;
    LS_S7_MoveBack2 : BOOL;
    LS_S7_MoveOut1 : BOOL;
    SOL_S2_Fix : BOOL;
    SOL_S7_Move1 : BOOL;
    LS_S7_MoveBack3 : BOOL;
    LS_S7_MoveBack4 : BOOL;
    SOL_S7_Move2 : BOOL;
    SOL_S7_Move3 : BOOL;
    SOL_S7_Move4 : BOOL;
    LS_S8_MoveBack : BOOL;
    SOL_S8_Move : BOOL;
    LS_S5_IndexFixBack : BOOL;
    SOL_S5_IndexFixBack : BOOL;
    SOL_S5_IndexFixOut : BOOL;
    LS_S6_IndexFixBack : BOOL;
    SOL_S6_IndexFixBack : BOOL;
    SOL_S6_IndexFixOut : BOOL;
    LS_S5_FixBack : BOOL;
    SOL_S5_Fix : BOOL;
    LS_S6_FixBack : BOOL;
    SOL_S6_Fix : BOOL;
    RY_Index : BOOL;
    HMIPB_SOL_IndexFixBack : BOOL;
    HMIPB_SOL_IndexFixOut : BOOL;
    AutoStatus : bool;
    LS_S5_IndexFixOut : BOOL;
    IndexCanRunStatus : bool;
    SystemReadyStatus : bool;
    ErrorStatus_MachineNonStop : bool;
    Error_LS_S5_IndexFixBack : BOOL;
    Error_LS_S5_IndexFixOut : BOOL;
    Error_SNR_Index : BOOL;
    Error_LS_S6_IndexFixBack : BOOL;
    Error_LS_S6_IndexFixOut : BOOL;
    HMIPB_RY_Index : BOOL;
    MaChineRunStatus : bool;
    LS_S6_IndexFixOut : BOOL;
    SNR_Index : BOOL;
    PB_Estop1 : BOOL;
    PB_Estop2 : BOOL;
    Error_PB_Estop1 : BOOL;
    Error_PB_Estop2 : BOOL;
    IndexData0 : StationRecord;
    IndexData2 : StationRecord;
    IndexData3 : StationRecord;
    IndexData5 : StationRecord;
    IndexData6 : StationRecord;
    IndexData7 : StationRecord;
    IndexData8 : StationRecord;
    HMIShow_OK2 : ARRAY[0..3] OF Bool;
    HMIShow_NG2 : ARRAY[0..3] OF Bool;
    HMIShow_OK3 : ARRAY[0..3] OF Bool;
    HMIShow_NG3 : ARRAY[0..3] OF Bool;
    HMIShow_OK5 : ARRAY[0..3] OF Bool;
    HMIShow_NG5 : ARRAY[0..3] OF Bool;
    HMIShow_OK6 : ARRAY[0..3] OF Bool;
    HMIShow_NG6 : ARRAY[0..3] OF Bool;
    HMIShow_OK7 : ARRAY[0..3] OF Bool;
    HMIShow_NG7 : ARRAY[0..3] OF Bool;
    HMIShow_OK8 : ARRAY[0..3] OF Bool;
    HMIShow_NG8 : ARRAY[0..3] OF Bool;
END_VAR
(*************************************************************************)
(******************************手動**************************************)
(*************************************************************************)
(*輸出IndexCanRunStatus*)
IndexCanRunStatus:=
(LS_S5_IndexFixOut AND NOT(SOL_S5_IndexFixBack) AND NOT(SOL_S5_IndexFixOut)) AND//S5Index
(LS_S6_IndexFixOut AND NOT(SOL_S6_IndexFixBack) AND NOT(SOL_S6_IndexFixOut)) AND//S6Index
(LS_S2_MoveBack AND NOT(SOL_S2_Move)) AND//S2
(LS_S3_MoveBack AND NOT(SOL_S3_Move)) AND//S3
(LS_S5_UpDownBack AND NOT(SOL_S5_UpDown) AND LS_S5_FixBack AND NOT(SOL_S5_Fix)) AND//S5
(LS_S6_UpDownBack AND NOT(SOL_S6_UpDown) AND LS_S6_FixBack AND NOT(SOL_S6_Fix)) AND//S6
(LS_S7_MoveBack1 AND LS_S7_MoveBack2 AND LS_S7_MoveBack3 AND LS_S7_MoveBack4 AND NOT(SOL_S7_Move1) AND NOT(SOL_S7_Move2) AND NOT(SOL_S7_Move3) AND NOT(SOL_S7_Move4)) AND //S7
(LS_S8_MoveBack AND NOT(SOL_S8_Move));//S8
(*轉盤運轉RY_Index*)
IF (AutoFlow=3 OR Autoflow=4) AND IndexCanRunStatus THEN
	RY_Index:=TRUE;
	ELSE
	RY_Index:=FALSE;
END_IF;

SOLIndexFixS5(
	inPushBackButton:=HMIPB_SOL_IndexFixBack,
	inPushOutButton:=HMIPB_SOL_IndexFixOut,
	inAutoStatus:=AutoStatus,
	inAutoFlowSet:=AutoFlow=2,
	inAutoFlowReset:=AutoFlow=6,
	inInterLockBack:=TRUE,
	inInterLockOut:=TRUE,
	inBackSensor:=LS_S5_IndexFixBack,
	inOutSensor:=LS_S5_IndexFixOut,
	outBackSol=>SOL_S5_IndexFixBack,
	outOutSol=>SOL_S5_IndexFixOut);
SOLIndexFixS6(
	inPushBackButton:=HMIPB_SOL_IndexFixBack,
	inPushOutButton:=HMIPB_SOL_IndexFixOut,
	inAutoStatus:=AutoStatus,
	inAutoFlowSet:=AutoFlow=2,
	inAutoFlowReset:=AutoFlow=6,
	inInterLockBack:=TRUE,
	inInterLockOut:=TRUE,
	inBackSensor:=LS_S6_IndexFixBack,
	inOutSensor:=LS_S6_IndexFixOut,
	outBackSol=>SOL_S6_IndexFixBack,
	outOutSol=>SOL_S6_IndexFixOut);
(*************************************************************************)
(*程序名稱:轉盤程式*)
(*作者:蔡相偉*)
(*版本,日期,版本資訊:*)
(*1.0.0	2017/8/8		初始版本*)
(*流程*)
(*PowerOn=0*)
(*Idle=1*)
(*轉盤定位出=2*)
(*轉盤起動=3*)
(*轉盤運轉中=4*)
(*轉盤停止=5*)
(*轉盤定位回=6*)
(*************************************************************************)
ErrorStatus:=
NOT(PB_Estop1) OR
NOT(PB_Estop2) OR
Error_PB_Estop1 OR
Error_PB_Estop2 OR
Error_SNR_Index OR
Error_LS_S5_IndexFixBack OR
Error_LS_S5_IndexFixOut OR
Error_LS_S6_IndexFixBack OR
Error_LS_S6_IndexFixOut;
(*PowerOn=0*)
IF NOT(SystemReadyStatus) OR ErrorStatus THEN
	AutoFlow:=0;
END_IF;
(*Idle=1*)
IF AutoFlow=0 AND SystemReadyStatus AND NOT(ErrorStatus) THEN
	AutoFlow:=1;
END_IF;
IF Autoflow=6 AND LS_S5_IndexFixBack AND LS_S6_IndexFixBack THEN
	Autoflow:=1;
END_IF;
(*轉盤定位出Turntable positioning out=2*)
R_TRIG_1(CLK:= HMIPB_RY_Index);
AllStationFinish:=
IndexData2.FinishFlag[2] AND
IndexData3.FinishFlag[3] AND
IndexData5.FinishFlag[5] AND
IndexData6.FinishFlag[6] AND
IndexData7.FinishFlag[7] AND
IndexData8.FinishFlag[8];

IF Autoflow=1 AND ((R_TRIG_1.Q AND NOT(AutoStatus)) OR
	(MachineRunStatus AND AutoStatus AND AllStationFinish)) THEN
	Autoflow:=2;
END_IF;
(*轉盤起動Turntable start=3*)
IF Autoflow=2 AND IndexCanRunStatus AND LS_S5_IndexFixOut AND LS_S6_IndexFixOut  THEN
	Autoflow:=3;
END_IF;
(*轉盤運轉中Turntable in operation=4*)
IF Autoflow=3 AND NOT(SNR_Index) THEN
	Autoflow:=4;
END_IF;
(*轉盤停止Turntable stop=5*)
IF Autoflow=4 AND SNR_Index THEN
	Autoflow:=5;
END_IF;
fIndexDataChange(EN:=AutoFlow=5);
(*轉盤定位回Turntable positioning back=6*)
IF Autoflow=5 THEN
	Autoflow:=6;
END_IF;
//**********************************************顯示
HMIShow_OK2[0]:=IndexData2.OKFlag_2[2] AND IndexData2.OKFlag_4[2];
HMIShow_NG2[0]:=IndexData2.NGFlag_2[2] OR IndexData2.NGFlag_4[2];

HMIShow_OK3[0]:=IndexData3.OKFlag_1[3] AND IndexData3.OKFlag_3[3];
HMIShow_NG3[0]:=IndexData3.NGFlag_1[3] OR IndexData3.NGFlag_3[3];

HMIShow_OK5[0]:=IndexData5.OKFlag_2[5];
HMIShow_OK5[1]:=IndexData5.OKFlag_4[5];
HMIShow_NG5[0]:=IndexData5.NGFlag_2[5];
HMIShow_NG5[1]:=IndexData5.NGFlag_4[5];

HMIShow_OK6[0]:=IndexData6.OKFlag_1[6];
HMIShow_OK6[1]:=IndexData6.OKFlag_3[6];
HMIShow_NG6[0]:=IndexData6.NGFlag_1[6];
HMIShow_NG6[1]:=IndexData6.NGFlag_3[6];

HMIShow_OK7[0]:=IndexData7.OKFlag_1[7];
HMIShow_OK7[1]:=IndexData7.OKFlag_2[7];
HMIShow_OK7[2]:=IndexData7.OKFlag_3[7];
HMIShow_OK7[3]:=IndexData7.OKFlag_4[7];
HMIShow_NG7[0]:=IndexData7.NGFlag_1[7];
HMIShow_NG7[1]:=IndexData7.NGFlag_2[7];
HMIShow_NG7[2]:=IndexData7.NGFlag_3[7];
HMIShow_NG7[3]:=IndexData7.NGFlag_4[7];

HMIShow_OK8[0]:=IndexData8.FinishFlag[8];
END_PROGRAM

PROGRAM prBowlFeeder
VAR
    bowlfedder1 : fbBowlFeeder;
    bowlfedder2 : fbBowlFeeder;
    bowlfedder3 : fbBowlFeeder;
    bowlfedder4 : fbBowlFeeder;
END_VAR
VAR_EXTERNAL
    HMI_ItemNotExistsDelayTime : ARRAY[0..6] OF LINT;
    HMI_ItemExistsDelayTime : ARRAY[0..6] OF LINT;
    HMI_ItemNotExistsErrorTime : ARRAY[0..6] OF LINT;
    SNR_S2_Full : BOOL;
    RY_S2_Full : BOOL;
    Error_SNR_S2_Full : BOOL;
    SNR_S3_Full : BOOL;
    RY_S3_Full : BOOL;
    Error_SNR_S3_Full : BOOL;
    SNR_S5_Full : BOOL;
    RY_S5_Full : BOOL;
    Error_SNR_S5_Full : BOOL;
    SNR_S6_Full : BOOL;
    RY_S6_Full : BOOL;
    Error_SNR_S6_Full : BOOL;
    RY_S2_Feed : BOOL;
    SOL_S2_Fix : BOOL;
    RY_S3_Feed : BOOL;
    SOL_S3_Fix : BOOL;
    RY_S5_Feed : BOOL;
    OutPutFeedRYS5 : BOOL;
    OutPutFeedRYS6 : BOOL;
    RY_S6_Feed : BOOL;
    LS_S2_THBack1 : BOOL;
    LS_S2_THBack2 : BOOL;
    SNR_S2_Feed : BOOL;
    LS_S3_THBack1 : BOOL;
    LS_S3_THBack2 : BOOL;
    SNR_S3_Feed : BOOL;
    FeedFlowS2 : INT;
    FeedFlowS3 : INT;
END_VAR
bowlfedder1(
	bFullSNR:=SNR_S2_Full,
	iItemNotExistDelayTime:=HMI_ItemNotExistsDelayTime[2],
	iItemExistTime:=HMI_ItemExistsDelayTime[2],
	iItemNotExistErrorTime:=HMI_ItemNotExistsErrorTime[2],
	bFullRY=>RY_S2_Full,
	bFullSNRError=>Error_SNR_S2_Full);
bowlfedder2(
	bFullSNR:=SNR_S3_Full,
	iItemNotExistDelayTime:=HMI_ItemNotExistsDelayTime[3],
	iItemExistTime:=HMI_ItemExistsDelayTime[3],
	iItemNotExistErrorTime:=HMI_ItemNotExistsErrorTime[3],
	bFullRY=>RY_S3_Full,
	bFullSNRError=>Error_SNR_S3_Full);
bowlfedder3(
	bFullSNR:=SNR_S5_Full,
	iItemNotExistDelayTime:=HMI_ItemNotExistsDelayTime[5],
	iItemExistTime:=HMI_ItemExistsDelayTime[5],
	iItemNotExistErrorTime:=HMI_ItemNotExistsErrorTime[5],
	bFullRY=>RY_S5_Full,
	bFullSNRError=>Error_SNR_S5_Full);
bowlfedder4(
	bFullSNR:=SNR_S6_Full,
	iItemNotExistDelayTime:=HMI_ItemNotExistsDelayTime[6],
	iItemExistTime:=HMI_ItemExistsDelayTime[6],
	iItemNotExistErrorTime:=HMI_ItemNotExistsErrorTime[6],
	bFullRY=>RY_S6_Full,
	bFullSNRError=>Error_SNR_S6_Full);
RY_S2_Feed:=RY_S2_Full OR FeedFlowS2>1;
RY_S3_Feed:=RY_S3_Full OR FeedFlowS3>1;
RY_S5_Feed:=RY_S5_Full OR OutPutFeedRYS5;
RY_S6_Feed:=RY_S6_Full OR OutPutFeedRYS6;
END_PROGRAM

PROGRAM prAxisDefineSt5L
VAR
    MC_Power1 : MC_Power;
    MC_Reset1 : MC_Reset;
    MC_Stop1 : MC_Stop;
    MC_Home1 : MC_Home;
    MC_TorqueControl1 : MC_TorqueControl;
    MC_TorqueControl2 : MC_TorqueControl;
    TorqueValue : LREAL;
    SpeedValue : LREAL;
    F_TRIG1 : F_TRIG;
    F_TRIG2 : F_TRIG;
    MC_MoveRelative1 : MC_MoveRelative;
    SpeedValue2 : LREAL;
    accdec : LREAL;
END_VAR
VAR_EXTERNAL CONSTANT
    _MC_ErrSta : WORD;
    MC_AxisLSt5 : _sAXIS_REF;
END_VAR
VAR_EXTERNAL
    HMIPB_ServoON_AxisLSt5 : BOOL;
    HMIPB_AlarmResetAxisLSt5 : BOOL;
    HMIPB_ServoStopAxisLSt5 : BOOL;
    HMIPB_SerchHome_AxisLSt5 : BOOL;
    PB_Reset1 : BOOL;
    PB_Reset2 : BOOL;
    PB_Estop1 : BOOL;
    PB_Estop2 : BOOL;
    HMI_ScrewTorque_St5_L : LREAL;
    HMI_ScrewSpeed_St5_L : LREAL;
    HMIPB_FW_AxisLSt5 : BOOL;
    HMIPB_RW_AxisLSt5 : BOOL;
    HMIShow_Homed : ARRAY[0..3] OF BOOL;
    HMIShow_Error : ARRAY[0..3] OF BOOL;
    HMIShow_POT : ARRAY[0..3] OF BOOL;
    HMIShow_NOT : ARRAY[0..3] OF BOOL;
    HMIShow_CurrentPosition : ARRAY[0..3] OF LREAL;
    HMIShow_CurrentSpeed : ARRAY[0..3] OF LREAL;
    HMIShow_CurrentTorque : ARRAY[0..3] OF LREAL;
    ScrewStartS5LFW : BOOL;
    ScrewStartS5LRW : BOOL;
    ResetAddress : ARRAY[0..3] OF bool;
    BackoutStart : ARRAY[0..3] OF BOOL;
    HMI_BackOutAngle_St5_L : LREAL;
    BackoutBusy : ARRAY[0..3] OF BOOL;
END_VAR
MC_Power1(Axis:=MC_AxisLSt5, Enable:=HMIPB_ServoON_AxisLSt5);		//servo on
MC_Reset1(Axis:=MC_AxisLSt5, Execute:=HMIPB_AlarmResetAxisLSt5 OR PB_Reset1 OR PB_Reset2);		//Alarm Reset
MC_Stop1(Axis:=MC_AxisLSt5, Execute:=NOT(PB_Estop1) OR NOT(PB_Estop2) OR HMIPB_ServoStopAxisLSt5 OR F_TRIG1.Q OR F_TRIG2.Q , Deceleration:=0, Jerk:=0, BufferMode:=_mcAborting);		//Servo Stop
MC_Home1(Axis:=MC_AxisLSt5, Execute:=HMIPB_SerchHome_AxisLSt5 OR ResetAddress[0]);		//Serch home
(*IF MC_Home1.Done OR MC_Home1.CommandAborted OR MC_Home1.Error THEN
	SerchHomeAxisS_InitialFlag:=FALSE;
END_IF;*)
TorqueValue:=HMI_ScrewTorque_St5_L;
SpeedValue:=HMI_ScrewSpeed_St5_L/360;
F_TRIG1(Clk:=HMIPB_FW_AxisLSt5 OR ScrewStartS5LFW);
F_TRIG2(Clk:=HMIPB_RW_AxisLSt5 OR ScrewStartS5LRW);
MC_TorqueControl1(Axis:=MC_AxisLSt5, Execute:=HMIPB_FW_AxisLSt5 OR ScrewStartS5LFW, Torque:=TorqueValue, TorqueRamp:=0, Velocity:=SpeedValue, Direction:=_mcPositiveDirection, BufferMode:=_mcAborting);		//JOG
MC_TorqueControl2(Axis:=MC_AxisLSt5, Execute:=HMIPB_RW_AxisLSt5 OR ScrewStartS5LRW, Torque:=TorqueValue, TorqueRamp:=0, Velocity:=SpeedValue, Direction:=_mcNegativeDirection, BufferMode:=_mcAborting);		//JOG
MC_MoveRelative1(Axis:=MC_AxisLSt5, Execute:=BackoutStart[0], Distance:=HMI_BackOutAngle_St5_L, Velocity:=HMI_ScrewSpeed_St5_L*2, Acceleration:=0, Deceleration:=0, Jerk:=0, BufferMode:=_mcAborting);
BackoutBusy[0]:=MC_MoveRelative1.Active;
//*****************************************************HMI Show**********************************************************************************************************
HMIShow_Homed[0]:=MC_AxisLSt5.Details.Homed;
HMIShow_Error[0]:=MC_AxisLSt5.DrvStatus.DrvAlarm OR MC_AxisLSt5.DrvStatus.DrvWarning OR NOT(MC_AxisLSt5.DrvStatus.MainPower) OR _MC_ErrSta<>0;
HMIShow_POT[0]:=NOT(MC_AxisLSt5.DrvStatus.P_OT);
HMIShow_NOT[0]:=NOT(MC_AxisLSt5.DrvStatus.N_OT);
HMIShow_CurrentPosition[0]:=MC_AxisLSt5.Act.Pos;
HMIShow_CurrentSpeed[0]:=MC_AxisLSt5.Act.Vel*360;
HMIShow_CurrentTorque[0]:=MC_AxisLSt5.Act.Trq;
END_PROGRAM

PROGRAM prAxisDefineSt5R
VAR
    MC_Power1 : MC_Power;
    MC_Reset1 : MC_Reset;
    MC_Stop1 : MC_Stop;
    MC_Home1 : MC_Home;
    MC_TorqueControl1 : MC_TorqueControl;
    MC_TorqueControl2 : MC_TorqueControl;
    TorqueValue : LREAL;
    SpeedValue : LREAL;
    F_TRIG1 : F_TRIG;
    F_TRIG2 : F_TRIG;
    MC_MoveRelative1 : MC_MoveRelative;
END_VAR
VAR_EXTERNAL CONSTANT
    _MC_ErrSta : WORD;
END_VAR
VAR_EXTERNAL
    PB_Reset1 : BOOL;
    PB_Reset2 : BOOL;
    PB_Estop1 : BOOL;
    PB_Estop2 : BOOL;
    HMIShow_Homed : ARRAY[0..3] OF BOOL;
    HMIShow_Error : ARRAY[0..3] OF BOOL;
    HMIShow_POT : ARRAY[0..3] OF BOOL;
    HMIShow_NOT : ARRAY[0..3] OF BOOL;
    HMIShow_CurrentPosition : ARRAY[0..3] OF LREAL;
    HMIShow_CurrentSpeed : ARRAY[0..3] OF LREAL;
    HMIShow_CurrentTorque : ARRAY[0..3] OF LREAL;
END_VAR
VAR_EXTERNAL CONSTANT
    MC_AxisRSt5 : _sAXIS_REF;
END_VAR
VAR_EXTERNAL
    HMIPB_ServoON_AxisRSt5 : BOOL;
    HMIPB_AlarmResetAxisRSt5 : BOOL;
    HMIPB_ServoStopAxisRSt5 : BOOL;
    HMIPB_SerchHome_AxisRSt5 : BOOL;
    HMI_ScrewTorque_St5_R : LREAL;
    HMI_ScrewSpeed_St5_R : LREAL;
    HMIPB_FW_AxisRSt5 : BOOL;
    HMIPB_RW_AxisRSt5 : BOOL;
    ScrewStartS5RFW : BOOL;
    ScrewStartS5RRW : BOOL;
    ResetAddress : ARRAY[0..3] OF bool;
    BackoutStart : ARRAY[0..3] OF BOOL;
    HMI_BackOutAngle_St5_R : LREAL;
    BackoutBusy : ARRAY[0..3] OF BOOL;
END_VAR
MC_Power1(Axis:=MC_AxisRSt5, Enable:=HMIPB_ServoON_AxisRSt5);		//servo on
MC_Reset1(Axis:=MC_AxisRSt5, Execute:=HMIPB_AlarmResetAxisRSt5 OR PB_Reset1 OR PB_Reset2);		//Alarm Reset
MC_Stop1(Axis:=MC_AxisRSt5, Execute:=NOT(PB_Estop1) OR NOT(PB_Estop2) OR HMIPB_ServoStopAxisRSt5 OR F_TRIG1.Q OR F_TRIG2.Q , Deceleration:=100, Jerk:=0, BufferMode:=_mcAborting);		//Servo Stop
MC_Home1(Axis:=MC_AxisRSt5, Execute:=HMIPB_SerchHome_AxisRSt5 OR ResetAddress[1]);		//Serch home
(*IF MC_Home1.Done OR MC_Home1.CommandAborted OR MC_Home1.Error THEN
	SerchHomeAxisS_InitialFlag:=FALSE;
END_IF;*)
TorqueValue:=HMI_ScrewTorque_St5_R;
SpeedValue:=HMI_ScrewSpeed_St5_R/360;
F_TRIG1(Clk:=HMIPB_FW_AxisRSt5 OR ScrewStartS5RFW);
F_TRIG2(Clk:=HMIPB_RW_AxisRSt5 OR ScrewStartS5RRW);
MC_TorqueControl1(Axis:=MC_AxisRSt5, Execute:=HMIPB_FW_AxisRSt5 OR ScrewStartS5RFW, Torque:=TorqueValue, TorqueRamp:=0, Velocity:=SpeedValue, Direction:=_mcPositiveDirection, BufferMode:=_mcAborting);		//JOG
MC_TorqueControl2(Axis:=MC_AxisRSt5, Execute:=HMIPB_RW_AxisRSt5 OR ScrewStartS5RRW, Torque:=TorqueValue, TorqueRamp:=0, Velocity:=SpeedValue, Direction:=_mcNegativeDirection, BufferMode:=_mcAborting);		//JOG
MC_MoveRelative1(Axis:=MC_AxisRSt5, Execute:=BackoutStart[1], Distance:=HMI_BackOutAngle_St5_R, Velocity:=HMI_ScrewSpeed_St5_R*2, Acceleration:=0, Deceleration:=0, Jerk:=0, BufferMode:=_mcAborting);
BackoutBusy[1]:=MC_MoveRelative1.Active;
//*****************************************************HMI Show**********************************************************************************************************
HMIShow_Homed[1]:=MC_AxisRSt5.Details.Homed;
HMIShow_Error[1]:=MC_AxisRSt5.DrvStatus.DrvAlarm OR MC_AxisRSt5.DrvStatus.DrvWarning OR NOT(MC_AxisRSt5.DrvStatus.MainPower) OR _MC_ErrSta<>0;
HMIShow_POT[1]:=NOT(MC_AxisRSt5.DrvStatus.P_OT);
HMIShow_NOT[1]:=NOT(MC_AxisRSt5.DrvStatus.N_OT);
HMIShow_CurrentPosition[1]:=MC_AxisRSt5.Act.Pos;
HMIShow_CurrentSpeed[1]:=MC_AxisRSt5.Act.Vel*360;
HMIShow_CurrentTorque[1]:=MC_AxisRSt5.Act.Trq;
END_PROGRAM

PROGRAM prAxisDefineSt6L
VAR
    MC_Power1 : MC_Power;
    MC_Reset1 : MC_Reset;
    MC_Stop1 : MC_Stop;
    MC_Home1 : MC_Home;
    MC_TorqueControl1 : MC_TorqueControl;
    MC_TorqueControl2 : MC_TorqueControl;
    TorqueValue : LREAL;
    SpeedValue : LREAL;
    F_TRIG1 : F_TRIG;
    F_TRIG2 : F_TRIG;
    MC_MoveRelative1 : MC_MoveRelative;
END_VAR
VAR_EXTERNAL CONSTANT
    _MC_ErrSta : WORD;
    MC_AxisLSt5 : _sAXIS_REF;
END_VAR
VAR_EXTERNAL
    HMIPB_ServoON_AxisLSt5 : BOOL;
    HMIPB_AlarmResetAxisLSt5 : BOOL;
    HMIPB_ServoStopAxisLSt5 : BOOL;
    HMIPB_SerchHome_AxisLSt5 : BOOL;
    PB_Reset1 : BOOL;
    PB_Reset2 : BOOL;
    PB_Estop1 : BOOL;
    PB_Estop2 : BOOL;
    HMI_ScrewTorque_St5_L : LREAL;
    HMI_ScrewSpeed_St5_L : LREAL;
    HMIPB_FW_AxisLSt5 : BOOL;
    HMIPB_RW_AxisLSt5 : BOOL;
    HMIShow_Homed : ARRAY[0..3] OF BOOL;
    HMIShow_Error : ARRAY[0..3] OF BOOL;
    HMIShow_POT : ARRAY[0..3] OF BOOL;
    HMIShow_NOT : ARRAY[0..3] OF BOOL;
    HMIShow_CurrentPosition : ARRAY[0..3] OF LREAL;
    HMIShow_CurrentSpeed : ARRAY[0..3] OF LREAL;
    HMIShow_CurrentTorque : ARRAY[0..3] OF LREAL;
END_VAR
VAR_EXTERNAL CONSTANT
    MC_AxisLSt6 : _sAXIS_REF;
END_VAR
VAR_EXTERNAL
    HMIPB_ServoON_AxisLSt6 : BOOL;
    HMIPB_AlarmResetAxisLSt6 : BOOL;
    HMIPB_ServoStopAxisLSt6 : BOOL;
    HMIPB_SerchHome_AxisLSt6 : BOOL;
    HMI_ScrewTorque_St6_L : LREAL;
    HMI_ScrewSpeed_St6_L : LREAL;
    HMIPB_FW_AxisLSt6 : BOOL;
    HMIPB_RW_AxisLSt6 : BOOL;
    ScrewStartS6LFW : BOOL;
    ScrewStartS6LRW : BOOL;
    ResetAddress : ARRAY[0..3] OF bool;
    BackoutStart : ARRAY[0..3] OF BOOL;
    HMI_BackOutAngle_St6_L : LREAL;
    BackoutBusy : ARRAY[0..3] OF BOOL;
END_VAR
MC_Power1(Axis:=MC_AxisLSt6, Enable:=HMIPB_ServoON_AxisLSt6);		//servo on
MC_Reset1(Axis:=MC_AxisLSt6, Execute:=HMIPB_AlarmResetAxisLSt6 OR PB_Reset1 OR PB_Reset2);		//Alarm Reset
MC_Stop1(Axis:=MC_AxisLSt6, Execute:=NOT(PB_Estop1) OR NOT(PB_Estop2) OR HMIPB_ServoStopAxisLSt6 OR F_TRIG1.Q OR F_TRIG2.Q , Deceleration:=100, Jerk:=0, BufferMode:=_mcAborting);		//Servo Stop
MC_Home1(Axis:=MC_AxisLSt6, Execute:=HMIPB_SerchHome_AxisLSt6 OR ResetAddress[2]);		//Serch home
(*IF MC_Home1.Done OR MC_Home1.CommandAborted OR MC_Home1.Error THEN
	SerchHomeAxisS_InitialFlag:=FALSE;
END_IF;*)
TorqueValue:=HMI_ScrewTorque_St6_L;
SpeedValue:=HMI_ScrewSpeed_St6_L/360;
F_TRIG1(Clk:=HMIPB_FW_AxisLSt6 OR ScrewStartS6LFW);
F_TRIG2(Clk:=HMIPB_RW_AxisLSt6 OR ScrewStartS6LRW);
MC_TorqueControl1(Axis:=MC_AxisLSt6, Execute:=HMIPB_FW_AxisLSt6 OR ScrewStartS6LFW, Torque:=TorqueValue, TorqueRamp:=0, Velocity:=SpeedValue, Direction:=_mcPositiveDirection, BufferMode:=_mcAborting);		//JOG
MC_TorqueControl2(Axis:=MC_AxisLSt6, Execute:=HMIPB_RW_AxisLSt6 OR ScrewStartS6LRW, Torque:=TorqueValue, TorqueRamp:=0, Velocity:=SpeedValue, Direction:=_mcNegativeDirection, BufferMode:=_mcAborting);		//JOG
MC_MoveRelative1(Axis:=MC_AxisLSt6, Execute:=BackoutStart[2], Distance:=HMI_BackOutAngle_St6_L, Velocity:=HMI_ScrewSpeed_St6_L*2, Acceleration:=0, Deceleration:=0, Jerk:=0, BufferMode:=_mcAborting);
BackoutBusy[2]:=MC_MoveRelative1.Active;
//*****************************************************HMI Show**********************************************************************************************************
HMIShow_Homed[2]:=MC_AxisLSt6.Details.Homed;
HMIShow_Error[2]:=MC_AxisLSt6.DrvStatus.DrvAlarm OR MC_AxisLSt6.DrvStatus.DrvWarning OR NOT(MC_AxisLSt6.DrvStatus.MainPower) OR _MC_ErrSta<>0;
HMIShow_POT[2]:=NOT(MC_AxisLSt6.DrvStatus.P_OT);
HMIShow_NOT[2]:=NOT(MC_AxisLSt6.DrvStatus.N_OT);
HMIShow_CurrentPosition[2]:=MC_AxisLSt6.Act.Pos;
HMIShow_CurrentSpeed[2]:=MC_AxisLSt6.Act.Vel*360;
HMIShow_CurrentTorque[2]:=MC_AxisLSt6.Act.Trq;
END_PROGRAM

PROGRAM prAxisDefineSt6R
VAR
    MC_Power1 : MC_Power;
    MC_Reset1 : MC_Reset;
    MC_Stop1 : MC_Stop;
    MC_Home1 : MC_Home;
    MC_TorqueControl1 : MC_TorqueControl;
    MC_TorqueControl2 : MC_TorqueControl;
    TorqueValue : LREAL;
    SpeedValue : LREAL;
    F_TRIG1 : F_TRIG;
    F_TRIG2 : F_TRIG;
    MC_MoveRelative1 : MC_MoveRelative;
END_VAR
VAR_EXTERNAL CONSTANT
    _MC_ErrSta : WORD;
END_VAR
VAR_EXTERNAL
    PB_Reset1 : BOOL;
    PB_Reset2 : BOOL;
    PB_Estop1 : BOOL;
    PB_Estop2 : BOOL;
    HMIShow_Homed : ARRAY[0..3] OF BOOL;
    HMIShow_Error : ARRAY[0..3] OF BOOL;
    HMIShow_POT : ARRAY[0..3] OF BOOL;
    HMIShow_NOT : ARRAY[0..3] OF BOOL;
    HMIShow_CurrentPosition : ARRAY[0..3] OF LREAL;
    HMIShow_CurrentSpeed : ARRAY[0..3] OF LREAL;
    HMIShow_CurrentTorque : ARRAY[0..3] OF LREAL;
END_VAR
VAR_EXTERNAL CONSTANT
    MC_AxisRSt6 : _sAXIS_REF;
END_VAR
VAR_EXTERNAL
    HMIPB_ServoON_AxisRSt6 : BOOL;
    HMIPB_AlarmResetAxisRSt6 : BOOL;
    HMIPB_ServoStopAxisRSt6 : BOOL;
    HMIPB_SerchHome_AxisRSt6 : BOOL;
    HMI_ScrewTorque_St6_R : LREAL;
    HMI_ScrewSpeed_St6_R : LREAL;
    HMIPB_FW_AxisRSt6 : BOOL;
    HMIPB_RW_AxisRSt6 : BOOL;
    ScrewStartS6RFW : BOOL;
    ScrewStartS6RRW : BOOL;
    ResetAddress : ARRAY[0..3] OF bool;
    BackoutStart : ARRAY[0..3] OF BOOL;
    HMI_BackOutAngle_St6_R : LREAL;
    BackoutBusy : ARRAY[0..3] OF BOOL;
END_VAR
MC_Power1(Axis:=MC_AxisRSt6, Enable:=HMIPB_ServoON_AxisRSt6);		//servo on
MC_Reset1(Axis:=MC_AxisRSt6, Execute:=HMIPB_AlarmResetAxisRSt6 OR PB_Reset1 OR PB_Reset2);		//Alarm Reset
MC_Stop1(Axis:=MC_AxisRSt6, Execute:=NOT(PB_Estop1) OR NOT(PB_Estop2) OR HMIPB_ServoStopAxisRSt6 OR F_TRIG1.Q OR F_TRIG2.Q , Deceleration:=100, Jerk:=0, BufferMode:=_mcAborting);		//Servo Stop
MC_Home1(Axis:=MC_AxisRSt6, Execute:=HMIPB_SerchHome_AxisRSt6 OR ResetAddress[3]);		//Serch home
(*IF MC_Home1.Done OR MC_Home1.CommandAborted OR MC_Home1.Error THEN
	SerchHomeAxisS_InitialFlag:=FALSE;
END_IF;*)
TorqueValue:=HMI_ScrewTorque_St6_R;
SpeedValue:=HMI_ScrewSpeed_St6_R/360;
F_TRIG1(Clk:=HMIPB_FW_AxisRSt6 OR ScrewStartS6RFW);
F_TRIG2(Clk:=HMIPB_RW_AxisRSt6 OR ScrewStartS6RRW);
MC_TorqueControl1(Axis:=MC_AxisRSt6, Execute:=HMIPB_FW_AxisRSt6 OR ScrewStartS6RFW, Torque:=TorqueValue, TorqueRamp:=0, Velocity:=SpeedValue, Direction:=_mcPositiveDirection, BufferMode:=_mcAborting);		//JOG
MC_TorqueControl2(Axis:=MC_AxisRSt6, Execute:=HMIPB_RW_AxisRSt6 OR ScrewStartS6RRW, Torque:=TorqueValue, TorqueRamp:=0, Velocity:=SpeedValue, Direction:=_mcNegativeDirection, BufferMode:=_mcAborting);		//JOG
MC_MoveRelative1(Axis:=MC_AxisRSt6, Execute:=BackoutStart[3], Distance:=HMI_BackOutAngle_St6_R, Velocity:=HMI_ScrewSpeed_St6_R*2, Acceleration:=0, Deceleration:=0, Jerk:=0, BufferMode:=_mcAborting);
BackoutBusy[3]:=MC_MoveRelative1.Active;
//*****************************************************HMI Show**********************************************************************************************************
HMIShow_Homed[3]:=MC_AxisRSt6.Details.Homed;
HMIShow_Error[3]:=MC_AxisRSt6.DrvStatus.DrvAlarm OR MC_AxisRSt6.DrvStatus.DrvWarning OR NOT(MC_AxisRSt6.DrvStatus.MainPower) OR _MC_ErrSta<>0;
HMIShow_POT[3]:=NOT(MC_AxisRSt6.DrvStatus.P_OT);
HMIShow_NOT[3]:=NOT(MC_AxisRSt6.DrvStatus.N_OT);
HMIShow_CurrentPosition[3]:=MC_AxisRSt6.Act.Pos;
HMIShow_CurrentSpeed[3]:=MC_AxisRSt6.Act.Vel*360;
HMIShow_CurrentTorque[3]:=MC_AxisRSt6.Act.Trq;
END_PROGRAM

PROGRAM prInitial
VAR
    Initflow : INT;
END_VAR
VAR_EXTERNAL
    SystemReadyStatus : bool;
    AutoStatus : bool;
END_VAR
IF P_First_Run THEN
	SystemReadyStatus:=FALSE;
	Initflow:=0;
END_IF;
IF Initflow=0 AND NOT(SystemReadyStatus) THEN
	Initflow:=1;
	SystemReadyStatus:=TRUE;
END_IF;
IF Initflow=1 AND SystemReadyStatus THEN
	AutoStatus:=TRUE;
	Initflow:=9999;
END_IF;
END_PROGRAM

PROGRAM prStation2
VAR
    SolMove : fbSingleSolRy;
    SolFix : fbSingleSolRy;
    SolTh1 : fbDoubleSolRy;
    SolTh2 : fbDoubleSolRy;
    ErrorState : BOOL;
    AutoFlow : INT;
    TON1 : TON;
    TON3OK : TON;
    TON3NG : TON;
    TON4 : TON;
    AutoFlowFeed : INT;
END_VAR
VAR RETAIN
    FeedFlag : BOOL;
END_VAR
VAR
    InitialFlow : INT;
    F_TRIG1 : F_TRIG;
    ErrorStateFeed : BOOL;
END_VAR
VAR_EXTERNAL
    AutoStatus : bool;
    SOL_S2_Move : BOOL;
    HMIPB_SOL_S2_Move : BOOL;
    HMIPB_SOL_S2_Fix : BOOL;
    LS_S2_THOut1 : BOOL;
    LS_S2_THOut2 : BOOL;
    SOL_S2_THBack1 : BOOL;
    SOL_S2_THBack2 : BOOL;
    SOL_S2_THOut1 : BOOL;
    SOL_S2_THOut2 : BOOL;
    SNR_Index : BOOL;
    SOL_S2_Fix : BOOL;
    LS_S2_THBack1 : BOOL;
    LS_S2_THBack2 : BOOL;
    HMIPB_SOL_S2_THBack1 : BOOL;
    HMIPB_SOL_S2_THOut1 : BOOL;
    HMIPB_SOL_S2_THBack2 : BOOL;
    HMIPB_SOL_S2_THOut2 : BOOL;
    LS_S2_MoveBack : BOOL;
    RY_Index : BOOL;
    IndexData2 : StationRecord;
    Error_PB_Estop1 : BOOL;
    Error_PB_Estop2 : BOOL;
    ErrorStatus_MachineNonStop : bool;
    Error_LS_S2_MoveBack : BOOL;
    Error_LS_S2_MoveOut : BOOL;
    Error_LS_S2_THBack1 : BOOL;
    Error_LS_S2_THBack2 : BOOL;
    Error_LS_S2_THOut1 : BOOL;
    Error_LS_S2_THOut2 : BOOL;
    SystemReadyStatus : bool;
    MachineRunStatus : bool;
    LS_S2_MoveOut : BOOL;
    SNR_S2_Feed : BOOL;
    Error_SNR_S2_Feed : BOOL;
    PB_Reset1 : BOOL;
    PB_Reset2 : BOOL;
    HMIPB_S2Feed : BOOL;
    HMIPB_DisableS2 : BOOL;
    FeedFlowS2 : INT;
    HMI_FeededS2 : BOOL;
END_VAR
SolMove(
	inPushButton:=HMIPB_SOL_S2_Move,
	inAutoStatus:=AutoStatus,
	inAutoFlowSet:=AutoFlow=3,
	inAutoFlowReset:=AutoFlow=4 OR ErrorState OR InitialFlow=2,
	inInterLockBack:=TRUE,
	inInterLockOut:=SNR_Index AND NOT(RY_Index) AND LS_S2_THOut1 AND LS_S2_THOut2 AND NOT(SOL_S2_THBack1) AND NOT(SOL_S2_THBack2) AND NOT(SOL_S2_THOut1) AND NOT(SOL_S2_THOut2),
	outSol=>SOL_S2_Move);
SolFix(
	inPushButton:=HMIPB_SOL_S2_Fix,
	inAutoStatus:=AutoStatus,
	inAutoFlowSet:=(AutoFlowFeed=3 OR AutoFlowFeed=6),
	inAutoFlowReset:=(AutoFlowFeed=4 OR AutoFlowFeed=7),
	inInterLockBack:=TRUE,
	inInterLockOut:=(LS_S2_THBack1 OR LS_S2_THOut1) AND LS_S2_THBack2 AND NOT(SOL_S2_THBack1) AND NOT(SOL_S2_THBack2) AND NOT(SOL_S2_THOut1) AND NOT(SOL_S2_THOut2),
	outSol=>SOL_S2_Fix);
SolTh1(
	inPushBackButton:=HMIPB_SOL_S2_THBack1,
	inPushOutButton:=HMIPB_SOL_S2_THOut1,
	inAutoStatus:=AutoStatus,
	inAutoFlowSet:=(AutoFlow=2 OR AutoFlowFeed=5),
	inAutoFlowReset:=AutoFlowFeed=2 OR InitialFlow=3,
	inInterLockBack:=LS_S2_MoveBack AND NOT(SOL_S2_Move),
	inInterLockOut:=LS_S2_MoveBack AND NOT(SOL_S2_Move) AND NOT(SOL_S2_Fix),
	inBackSensor:=LS_S2_THBack1,
	inOutSensor:=LS_S2_THOut1,
	outBackSol=>SOL_S2_THBack1,
	outOutSol=>SOL_S2_THOut1);
SolTh2(
	inPushBackButton:=HMIPB_SOL_S2_THBack2,
	inPushOutButton:=HMIPB_SOL_S2_THOut2,
	inAutoStatus:=AutoStatus,
	inAutoFlowSet:=AutoFlow=2,
	inAutoFlowReset:=AutoFlowFeed=2 OR InitialFlow=3,
	inInterLockBack:=LS_S2_MoveBack AND NOT(SOL_S2_Move),
	inInterLockOut:=LS_S2_MoveBack AND NOT(SOL_S2_Move) AND NOT(SOL_S2_Fix),
	inBackSensor:=LS_S2_THBack2,
	inOutSensor:=LS_S2_THOut2,
	outBackSol=>SOL_S2_THBack2,
	outOutSol=>SOL_S2_THOut2);
(*************************************************************************************************************)
(*EStOP and Error*)
IF (Error_PB_Estop1 OR Error_PB_Estop2) AND NOT(IndexData2.OKFlag_4[2]) THEN
	IndexData2.NGFlag_4[2]:=TRUE;
	IndexData2.ErrorRecordData[2]:=1;
END_IF;
IF (Error_PB_Estop1 OR Error_PB_Estop2) AND NOT(IndexData2.OKFlag_2[2]) THEN
	IndexData2.NGFlag_2[2]:=TRUE;
	IndexData2.ErrorRecordData[2]:=1;
END_IF;
IF ErrorState AND NOT(IndexData2.OKFlag_4[2]) THEN
	IndexData2.NGFlag_4[2]:=TRUE;
	IndexData2.ErrorRecordData[2]:=2;
END_IF;
IF ErrorState AND NOT(IndexData2.OKFlag_2[2])  THEN
	IndexData2.NGFlag_2[2]:=TRUE;
	IndexData2.ErrorRecordData[2]:=2;
END_IF;
(*本站停工*)
IF HMIPB_DisableS2 AND NOT(IndexData2.FinishFlag[2]) THEN
	IndexData2.NGFlag_4[2]:=TRUE;
	IndexData2.NGFlag_2[2]:=TRUE;
END_IF;
(*本站狀態判斷*)
IF (IndexData2.OKFlag_4[2] OR IndexData2.NGFlag_4[2]) AND (IndexData2.OKFlag_2[2] OR IndexData2.NGFlag_2[2]) THEN
	IndexData2.FinishFlag[2]:=TRUE;
END_IF;
(*異常*)
ErrorState:=
Error_LS_S2_MoveBack OR
Error_LS_S2_MoveOut OR
ErrorStateFeed;
//*********************************自動********************************************
//****************************power on=0
IF NOT(SystemReadyStatus) OR ErrorState OR Error_PB_Estop1 OR Error_PB_Estop2 OR NOT(AutoStatus) THEN
	Autoflow:=0;
END_IF;

//*******************************idle=1
IF AutoFlow=0 AND NOT(NOT(SystemReadyStatus) OR ErrorState OR Error_PB_Estop1 OR Error_PB_Estop2 OR NOT(AutoStatus)) THEN
	AutoFlow:=1;
END_IF;
IF AutoFlow=4 AND HMIPB_S2Feed AND LS_S2_MoveBack THEN
	AutoFlow:=1;
END_IF;

//*******************************節流出=2
IF AutoFlow=1 AND
	HMI_FeededS2 AND
	MachineRunStatus AND
	NOT(IndexData2.FinishFlag[2]) THEN
	AutoFlow:=2;
END_IF;

//*******************************推出=3
IF AutoFlow=2 AND LS_S2_THOut1 AND LS_S2_THOut2 THEN
	AutoFlow:=3;
	HMI_FeededS2:=FALSE;
END_IF;
TON1(In:=AutoFlow=3 AND LS_S2_MoveOut, PT:=t#1s);
//*******************************推回=4
IF AutoFlow=3 AND TON1.Q THEN
	AutoFlow:=4;
	IndexData2.OKFlag_4[2]:=TRUE;
	IndexData2.OKFlag_2[2]:=TRUE;
	HMIPB_S2Feed:=TRUE;
END_IF;

//*********************************取料********************************************
(*異常*)
ErrorStateFeed:=
Error_LS_S2_THBack1 OR
Error_LS_S2_THBack2 OR
Error_LS_S2_THOut1 OR
Error_LS_S2_THOut2;
//****************************power on=0
IF NOT(SystemReadyStatus) OR ErrorStateFeed OR Error_PB_Estop1 OR Error_PB_Estop2 THEN
	AutoFlowFeed:=0;
END_IF;
//****************************idle=1
IF AutoFlowFeed=0 AND NOT(NOT(SystemReadyStatus) OR ErrorStateFeed OR Error_PB_Estop1 OR Error_PB_Estop2) THEN
	AutoFlowFeed:=1;
END_IF;
IF AutoFlowFeed=7 AND NOT(HMIPB_S2Feed) THEN
	AutoFlowFeed:=1;
END_IF;
//****************************節流回=2
IF AutoFlowFeed=1 AND HMIPB_S2Feed AND NOT(HMIPB_DisableS2) THEN
	AutoFlowFeed:=2;
END_IF;
//****************************擋料出=3
IF AutoFlowFeed=2 AND LS_S2_THBack1 AND LS_S2_THBack2 THEN
	AutoFlowFeed:=3;
END_IF;
TON3OK(In:=(AutoFlowFeed=3 OR AutoFlowFeed=6) AND SOL_S2_Fix AND SNR_S2_Feed, PT:=t#300ms);
TON3NG(In:=(AutoFlowFeed=3 OR AutoFlowFeed=6) AND SOL_S2_Fix AND NOT(SNR_S2_Feed), PT:=t#2s);
IF TON3NG.Q THEN
	Error_SNR_S2_Feed:=TRUE;
END_IF;
IF PB_Reset1 OR PB_Reset2 THEN
	Error_SNR_S2_Feed:=FALSE;
END_IF;
//****************************擋料回=4
IF AutoFlowFeed=3 AND (TON3OK.Q OR TON3NG.Q) AND NOT(Error_SNR_S2_Feed) THEN
	AutoFlowFeed:=4;
END_IF;
TON4(In:=AutoFlowFeed=4 AND NOT(SOL_S2_Fix), PT:=t#300ms);
//****************************節流1出=5
IF AutoFlowFeed=4 AND TON4.Q THEN
	AutoFlowFeed:=5;
END_IF;
//****************************擋料出=6
IF AutoFlowFeed=5 AND LS_S2_THOut1 THEN
	AutoFlowFeed:=6;
END_IF;
//****************************擋料回=7
IF AutoFlowFeed=6 AND (TON3OK.Q OR TON3NG.Q) AND NOT(Error_SNR_S2_Feed) THEN
	AutoFlowFeed:=7;
	HMI_FeededS2:=TRUE;
	HMIPB_S2Feed:=FALSE;
END_IF;
FeedFlowS2:=AutoFlowFeed;
//*********************************復歸********************************************
//****************************power on=0
IF NOT(SystemReadyStatus) THEN
	InitialFlow:=0;
END_IF;
//****************************idle=1
IF InitialFlow=0 AND (SystemReadyStatus) THEN
	InitialFlow:=1;
END_IF;
IF InitialFlow=3 AND LS_S2_THBack1 AND LS_S2_THBack2 THEN
	InitialFlow:=1;
END_IF;
//****************************推回=2
F_TRIG1(Clk:=ErrorStateFeed);
IF InitialFlow=1 AND F_TRIG1.Q THEN
	InitialFlow:=2;
END_IF;
//****************************節流回=3
IF InitialFlow=2 AND LS_S2_MoveBack THEN
	InitialFlow:=3;
END_IF;
END_PROGRAM

PROGRAM prStation3
VAR
    SolMove : fbSingleSolRy;
    SolFix : fbSingleSolRy;
    SolTh1 : fbDoubleSolRy;
    SolTh2 : fbDoubleSolRy;
    ErrorState : BOOL;
    TON1 : TON;
    Autoflow : INT;
    ErrorStateFeed : BOOL;
    AutoFlowFeed : INT;
    TON3OK : TON;
    TON3NG : TON;
    TON4 : TON;
END_VAR
VAR RETAIN
    FeedFlag : BOOL;
END_VAR
VAR
    InitialFlow : INT;
    F_TRIG1 : F_TRIG;
END_VAR
VAR_EXTERNAL
    AutoStatus : bool;
    SOL_S2_Move : BOOL;
    HMIPB_SOL_S2_Move : BOOL;
    HMIPB_SOL_S2_Fix : BOOL;
    LS_S2_THOut1 : BOOL;
    LS_S2_THOut2 : BOOL;
    SOL_S2_THBack1 : BOOL;
    SOL_S2_THBack2 : BOOL;
    SOL_S2_THOut1 : BOOL;
    SOL_S2_THOut2 : BOOL;
    SNR_Index : BOOL;
    SOL_S2_Fix : BOOL;
    LS_S2_THBack1 : BOOL;
    LS_S2_THBack2 : BOOL;
    HMIPB_SOL_S2_THBack1 : BOOL;
    HMIPB_SOL_S2_THOut1 : BOOL;
    HMIPB_SOL_S2_THBack2 : BOOL;
    HMIPB_SOL_S2_THOut2 : BOOL;
    LS_S2_MoveBack : BOOL;
    HMIPB_SOL_S3_Move : BOOL;
    LS_S3_THOut1 : BOOL;
    LS_S3_THOut2 : BOOL;
    SOL_S3_THBack1 : BOOL;
    SOL_S3_THBack2 : BOOL;
    SOL_S3_THOut1 : BOOL;
    SOL_S3_THOut2 : BOOL;
    SOL_S3_Move : BOOL;
    HMIPB_SOL_S3_Fix : BOOL;
    LS_S3_THBack1 : BOOL;
    LS_S3_THBack2 : BOOL;
    SOL_S3_Fix : BOOL;
    HMIPB_SOL_S3_THBack1 : BOOL;
    HMIPB_SOL_S3_THOut1 : BOOL;
    LS_S3_MoveBack : BOOL;
    HMIPB_SOL_S3_THBack2 : BOOL;
    HMIPB_SOL_S3_THOut2 : BOOL;
    RY_Index : BOOL;
    Error_PB_Estop1 : BOOL;
    Error_PB_Estop2 : BOOL;
    IndexData3 : StationRecord;
    Error_LS_S3_MoveBack : BOOL;
    Error_LS_S3_MoveOut : BOOL;
    SystemReadyStatus : bool;
    HMIPB_S3Feed : BOOL;
    MachineRunStatus : bool;
    LS_S3_MoveOut : BOOL;
    Error_LS_S3_THBack1 : BOOL;
    Error_LS_S3_THBack2 : BOOL;
    Error_LS_S3_THOut1 : BOOL;
    Error_LS_S3_THOut2 : BOOL;
    SNR_S3_Feed : BOOL;
    Error_SNR_S3_Feed : BOOL;
    PB_Reset1 : BOOL;
    PB_Reset2 : BOOL;
    HMIPB_DisableS3 : BOOL;
    FeedFlowS3 : INT;
    HMI_FeededS3 : BOOL;
END_VAR
SolMove(
	inPushButton:=HMIPB_SOL_S3_Move,
	inAutoStatus:=AutoStatus,
	inAutoFlowSet:=AutoFlow=3,
	inAutoFlowReset:=AutoFlow=4 OR ErrorState OR InitialFlow=2,
	inInterLockBack:=TRUE,
	inInterLockOut:=SNR_Index AND NOT(RY_Index) AND LS_S3_THOut1 AND LS_S3_THOut2 AND NOT(SOL_S3_THBack1) AND NOT(SOL_S3_THBack2) AND NOT(SOL_S3_THOut1) AND NOT(SOL_S3_THOut2),
	outSol=>SOL_S3_Move);
SolFix(
	inPushButton:=HMIPB_SOL_S3_Fix,
	inAutoStatus:=AutoStatus,
	inAutoFlowSet:=(AutoFlowFeed=3 OR AutoFlowFeed=6),
	inAutoFlowReset:=(AutoFlowFeed=4 OR AutoFlowFeed=7),
	inInterLockBack:=TRUE,
	inInterLockOut:=(LS_S3_THBack1 OR LS_S3_THOut1) AND LS_S3_THBack2 AND NOT(SOL_S3_THBack1) AND NOT(SOL_S3_THBack2) AND NOT(SOL_S3_THOut1) AND NOT(SOL_S3_THOut2),
	outSol=>SOL_S3_Fix);
SolTh1(
	inPushBackButton:=HMIPB_SOL_S3_THBack1,
	inPushOutButton:=HMIPB_SOL_S3_THOut1,
	inAutoStatus:=AutoStatus,
	inAutoFlowSet:=(AutoFlow=2 OR AutoFlowFeed=5),
	inAutoFlowReset:=AutoFlowFeed=2 OR InitialFlow=3,
	inInterLockBack:=LS_S3_MoveBack AND NOT(SOL_S3_Move),
	inInterLockOut:=LS_S3_MoveBack AND NOT(SOL_S3_Move) AND NOT(SOL_S3_Fix),
	inBackSensor:=LS_S3_THBack1,
	inOutSensor:=LS_S3_THOut1,
	outBackSol=>SOL_S3_THBack1,
	outOutSol=>SOL_S3_THOut1);
SolTh2(
	inPushBackButton:=HMIPB_SOL_S3_THBack2,
	inPushOutButton:=HMIPB_SOL_S3_THOut2,
	inAutoStatus:=AutoStatus,
	inAutoFlowSet:=AutoFlow=2,
	inAutoFlowReset:=AutoFlowFeed=2 OR InitialFlow=3,
	inInterLockBack:=LS_S3_MoveBack AND NOT(SOL_S3_Move),
	inInterLockOut:=LS_S3_MoveBack AND NOT(SOL_S3_Move) AND NOT(SOL_S3_Fix),
	inBackSensor:=LS_S3_THBack2,
	inOutSensor:=LS_S3_THOut2,
	outBackSol=>SOL_S3_THBack2,
	outOutSol=>SOL_S3_THOut2);
(*************************************************************************************************************)
(*EStOP and Error*)
IF (Error_PB_Estop1 OR Error_PB_Estop2) AND NOT(IndexData3.OKFlag_3[3]) THEN
	IndexData3.NGFlag_3[3]:=TRUE;
	IndexData3.ErrorRecordData[3]:=1;
END_IF;
IF (Error_PB_Estop1 OR Error_PB_Estop2) AND NOT(IndexData3.OKFlag_1[3]) THEN
	IndexData3.NGFlag_1[3]:=TRUE;
	IndexData3.ErrorRecordData[3]:=1;
END_IF;
IF ErrorState AND NOT(IndexData3.OKFlag_3[3]) THEN
	IndexData3.NGFlag_3[3]:=TRUE;
	IndexData3.ErrorRecordData[3]:=2;
END_IF;
IF ErrorState AND NOT(IndexData3.OKFlag_1[3]) THEN
	IndexData3.NGFlag_1[3]:=TRUE;
	IndexData3.ErrorRecordData[3]:=2;
END_IF;
(*本站停工*)
IF HMIPB_DisableS3 AND NOT(IndexData3.FinishFlag[3]) THEN
	IndexData3.NGFlag_3[3]:=TRUE;
	IndexData3.NGFlag_1[3]:=TRUE;
END_IF;
(*本站狀態判斷*)
IF (IndexData3.OKFlag_3[3] OR IndexData3.NGFlag_3[3]) AND (IndexData3.OKFlag_1[3] OR IndexData3.NGFlag_1[3]) THEN
	IndexData3.FinishFlag[3]:=TRUE;
END_IF;
(*異常*)
ErrorState:=
Error_LS_S3_MoveBack OR
Error_LS_S3_MoveOut OR
ErrorStateFeed;
//*********************************自動********************************************
//****************************power on=0
IF NOT(SystemReadyStatus) OR ErrorState OR Error_PB_Estop1 OR Error_PB_Estop2 OR NOT(AutoStatus) THEN
	Autoflow:=0;
END_IF;

//*******************************idle=1
IF AutoFlow=0 AND NOT(NOT(SystemReadyStatus) OR ErrorState OR Error_PB_Estop1 OR Error_PB_Estop2 OR NOT(AutoStatus)) THEN
	AutoFlow:=1;
END_IF;
IF AutoFlow=4 AND HMIPB_S3Feed AND LS_S3_MoveBack THEN
	AutoFlow:=1;
END_IF;

//*******************************節流出=2
IF AutoFlow=1 AND
	HMI_FeededS3 AND
	MachineRunStatus AND
	NOT(IndexData3.FinishFlag[3]) THEN
	AutoFlow:=2;
END_IF;

//*******************************推出=3
IF AutoFlow=2 AND LS_S3_THOut1 AND LS_S3_THOut2 THEN
	AutoFlow:=3;
	HMI_FeededS3:=FALSE;
END_IF;
TON1(In:=AutoFlow=3 AND LS_S3_MoveOut, PT:=t#1s);
//*******************************推回=4
IF AutoFlow=3 AND TON1.Q THEN
	AutoFlow:=4;
	IndexData3.OKFlag_3[3]:=TRUE;
	IndexData3.OKFlag_1[3]:=TRUE;
	HMIPB_S3Feed:=TRUE;
END_IF;

//*********************************取料********************************************
(*異常*)
ErrorStateFeed:=
Error_LS_S3_THBack1 OR
Error_LS_S3_THBack2 OR
Error_LS_S3_THOut1 OR
Error_LS_S3_THOut2;
//****************************power on=0
IF NOT(SystemReadyStatus) OR ErrorStateFeed OR Error_PB_Estop1 OR Error_PB_Estop2 THEN
	AutoFlowFeed:=0;
END_IF;
//****************************idle=1
IF AutoFlowFeed=0 AND NOT(NOT(SystemReadyStatus) OR ErrorStateFeed OR Error_PB_Estop1 OR Error_PB_Estop2) THEN
	AutoFlowFeed:=1;
END_IF;
IF AutoFlowFeed=7 AND NOT(HMIPB_S3Feed) THEN
	AutoFlowFeed:=1;
END_IF;
//****************************節流回=2
IF AutoFlowFeed=1 AND HMIPB_S3Feed THEN
	AutoFlowFeed:=2;
END_IF;
//****************************擋料出=3
IF AutoFlowFeed=2 AND LS_S3_THBack1 AND LS_S3_THBack2 THEN
	AutoFlowFeed:=3;
END_IF;
TON3OK(In:=(AutoFlowFeed=3 OR AutoFlowFeed=6) AND SOL_S3_Fix AND SNR_S3_Feed, PT:=t#300ms);
TON3NG(In:=(AutoFlowFeed=3 OR AutoFlowFeed=6) AND SOL_S3_Fix AND NOT(SNR_S3_Feed), PT:=t#2s);
IF TON3NG.Q THEN
	Error_SNR_S3_Feed:=TRUE;
END_IF;
IF PB_Reset1 OR PB_Reset2 THEN
	Error_SNR_S3_Feed:=FALSE;
END_IF;
//****************************擋料回=4
IF AutoFlowFeed=3 AND (TON3OK.Q OR TON3NG.Q) AND NOT(Error_SNR_S3_Feed) THEN
	AutoFlowFeed:=4;
END_IF;
TON4(In:=AutoFlowFeed=4 AND NOT(SOL_S3_Fix), PT:=t#300ms);
//****************************節流1出=5
IF AutoFlowFeed=4 AND TON4.Q THEN
	AutoFlowFeed:=5;
END_IF;
//****************************擋料出=6
IF AutoFlowFeed=5 AND LS_S3_THOut1 THEN
	AutoFlowFeed:=6;
END_IF;
//****************************擋料回=7
IF AutoFlowFeed=6 AND (TON3OK.Q OR TON3NG.Q) AND NOT(Error_SNR_S3_Feed) THEN
	AutoFlowFeed:=7;
	HMI_FeededS3:=TRUE;
	HMIPB_S3Feed:=FALSE;
END_IF;
FeedFlowS3:=AutoFlowFeed;
//*********************************復歸********************************************
//****************************power on=0
IF NOT(SystemReadyStatus) THEN
	InitialFlow:=0;
END_IF;
//****************************idle=1
IF InitialFlow=0 AND (SystemReadyStatus) THEN
	InitialFlow:=1;
END_IF;
IF InitialFlow=3 AND LS_S3_THBack1 AND LS_S3_THBack2 THEN
	InitialFlow:=1;
END_IF;
//****************************推回=2
F_TRIG1(Clk:=ErrorStateFeed);
IF InitialFlow=1 AND F_TRIG1.Q THEN
	InitialFlow:=2;
END_IF;
//****************************節流回=3
IF InitialFlow=2 AND LS_S3_MoveBack THEN
	InitialFlow:=3;
END_IF;
END_PROGRAM

PROGRAM prStation7
VAR
    SolMove1 : fbSingleSolRy;
    SolMove2 : fbSingleSolRy;
    SolMove3 : fbSingleSolRy;
    SolMove4 : fbSingleSolRy;
    ErrorState : BOOL;
    Autoflow : INT;
    pushFlag1 : BOOL;
    pushFlag2 : BOOL;
    pushFlag3 : BOOL;
    pushFlag4 : BOOL;
    TON1 : TON;
    RTRIG1 : R_TRIG;
    RTRIG2 : R_TRIG;
    RTRIG3 : R_TRIG;
    RTRIG4 : R_TRIG;
END_VAR
VAR_EXTERNAL
    HMIPB_SOL_S7_Move1 : BOOL;
    AutoStatus : bool;
    SNR_Index : BOOL;
    RY_Index : BOOL;
    SOL_S7_Move1 : BOOL;
    HMIPB_SOL_S7_Move2 : BOOL;
    SOL_S7_Move2 : BOOL;
    HMIPB_SOL_S7_Move3 : BOOL;
    SOL_S7_Move3 : BOOL;
    HMIPB_SOL_S7_Move4 : BOOL;
    SOL_S7_Move4 : BOOL;
    Error_PB_Estop1 : BOOL;
    Error_PB_Estop2 : BOOL;
    IndexData7 : StationRecord;
    Error_LS_S7_MoveBack1 : BOOL;
    Error_LS_S7_MoveOut1 : BOOL;
    Error_LS_S7_MoveBack2 : BOOL;
    Error_LS_S7_MoveOut2 : BOOL;
    Error_LS_S7_MoveBack3 : BOOL;
    Error_LS_S7_MoveOut3 : BOOL;
    Error_LS_S7_MoveOut4 : BOOL;
    Error_LS_S7_MoveBack4 : BOOL;
    SystemReadyStatus : bool;
    MachineRunStatus : bool;
    LS_S7_MoveOut1 : BOOL;
    LS_S7_MoveOut2 : BOOL;
    LS_S7_MoveOut3 : BOOL;
    LS_S7_MoveOut4 : BOOL;
    LS_S7_MoveBack1 : BOOL;
    LS_S7_MoveBack2 : BOOL;
    LS_S7_MoveBack3 : BOOL;
    LS_S7_MoveBack4 : BOOL;
    OKCount : UDINT;
    TotalCount : UDINT;
END_VAR
SolMove1(
	inPushButton:=HMIPB_SOL_S7_Move1,
	inAutoStatus:=AutoStatus,
	inAutoFlowSet:=pushFlag1,
	inAutoFlowReset:=Autoflow=4 OR ErrorState,
	inInterLockBack:=TRUE,
	inInterLockOut:=SNR_Index AND NOT(RY_Index),
	outSol=>SOL_S7_Move1);
SolMove2(
	inPushButton:=HMIPB_SOL_S7_Move2,
	inAutoStatus:=AutoStatus,
	inAutoFlowSet:=pushFlag2,
	inAutoFlowReset:=Autoflow=4 OR ErrorState,
	inInterLockBack:=TRUE,
	inInterLockOut:=SNR_Index AND NOT(RY_Index),
	outSol=>SOL_S7_Move2);
SolMove3(
	inPushButton:=HMIPB_SOL_S7_Move3,
	inAutoStatus:=AutoStatus,
	inAutoFlowSet:=pushFlag3,
	inAutoFlowReset:=Autoflow=4 OR ErrorState,
	inInterLockBack:=TRUE,
	inInterLockOut:=SNR_Index AND NOT(RY_Index),
	outSol=>SOL_S7_Move3);
SolMove4(
	inPushButton:=HMIPB_SOL_S7_Move4,
	inAutoStatus:=AutoStatus,
	inAutoFlowSet:=pushFlag4,
	inAutoFlowReset:=Autoflow=4 OR ErrorState,
	inInterLockBack:=TRUE,
	inInterLockOut:=SNR_Index AND NOT(RY_Index),
	outSol=>SOL_S7_Move4);
(*************************************************************************************************************)
(*EStOP and Error*)
IF (Error_PB_Estop1 OR Error_PB_Estop2) AND NOT(IndexData7.OKFlag_1[7]) THEN
	IndexData7.NGFlag_1[7]:=TRUE;
	IndexData7.ErrorRecordData[7]:=1;
END_IF;
IF (Error_PB_Estop1 OR Error_PB_Estop2) AND NOT(IndexData7.OKFlag_2[7]) THEN
	IndexData7.NGFlag_2[7]:=TRUE;
	IndexData7.ErrorRecordData[7]:=1;
END_IF;
IF (Error_PB_Estop1 OR Error_PB_Estop2) AND NOT(IndexData7.OKFlag_3[7]) THEN
	IndexData7.NGFlag_3[7]:=TRUE;
	IndexData7.ErrorRecordData[7]:=1;
END_IF;
IF (Error_PB_Estop1 OR Error_PB_Estop2) AND NOT(IndexData7.OKFlag_4[7]) THEN
	IndexData7.NGFlag_4[7]:=TRUE;
	IndexData7.ErrorRecordData[7]:=1;
END_IF;
IF (Error_LS_S7_MoveBack1 OR Error_LS_S7_MoveOut1) AND NOT(IndexData7.OKFlag_1[7]) THEN
	IndexData7.NGFlag_1[7]:=TRUE;
	IndexData7.ErrorRecordData[7]:=2;
END_IF;
IF (Error_LS_S7_MoveBack2 OR Error_LS_S7_MoveOut2) AND NOT(IndexData7.OKFlag_2[7]) THEN
	IndexData7.NGFlag_2[7]:=TRUE;
	IndexData7.ErrorRecordData[7]:=2;
END_IF;
IF (Error_LS_S7_MoveBack3 OR Error_LS_S7_MoveOut3) AND NOT(IndexData7.OKFlag_3[7]) THEN
	IndexData7.NGFlag_3[7]:=TRUE;
	IndexData7.ErrorRecordData[7]:=2;
END_IF;
IF (Error_LS_S7_MoveBack4 OR Error_LS_S7_MoveOut4) AND NOT(IndexData7.OKFlag_4[7]) THEN
	IndexData7.NGFlag_4[7]:=TRUE;
	IndexData7.ErrorRecordData[7]:=2;
END_IF;
(*本站狀態判斷*)
IF (IndexData7.OKFlag_1[7] OR IndexData7.NGFlag_1[7]) AND
	(IndexData7.OKFlag_2[7] OR IndexData7.NGFlag_2[7]) AND
	(IndexData7.OKFlag_3[7] OR IndexData7.NGFlag_3[7]) AND
	(IndexData7.OKFlag_4[7] OR IndexData7.NGFlag_4[7])
	THEN
	IndexData7.FinishFlag[7]:=TRUE;
END_IF;
(*前站判斷*)
IF IndexData7.NGFlag_1[6] OR NOT(IndexData7.OKFlag_1[6]) THEN
	IndexData7.NGFlag_1[7]:=TRUE;
END_IF;
IF IndexData7.NGFlag_3[6] OR NOT(IndexData7.OKFlag_3[6]) THEN
	IndexData7.NGFlag_3[7]:=TRUE;
END_IF;
IF IndexData7.NGFlag_2[5] OR NOT(IndexData7.OKFlag_2[5]) THEN
	IndexData7.NGFlag_2[7]:=TRUE;
END_IF;
IF IndexData7.NGFlag_4[5] OR NOT(IndexData7.OKFlag_4[5]) THEN
	IndexData7.NGFlag_4[7]:=TRUE;
END_IF;
(*異常*)
ErrorState:=
Error_LS_S7_MoveBack1 OR
Error_LS_S7_MoveOut1 OR
Error_LS_S7_MoveBack2 OR
Error_LS_S7_MoveOut2 OR
Error_LS_S7_MoveBack3 OR
Error_LS_S7_MoveOut3 OR
Error_LS_S7_MoveBack4 OR
Error_LS_S7_MoveOut4;
IF ErrorState THEN
	pushFlag1:=FALSE;
	pushFlag2:=FALSE;
	pushFlag3:=FALSE;
	pushFlag4:=FALSE;
END_IF;
//*********************************自動********************************************
//****************************power on=0
IF NOT(SystemReadyStatus) OR ErrorState OR Error_PB_Estop1 OR Error_PB_Estop2 OR NOT(AutoStatus) THEN
	Autoflow:=0;
END_IF;

//*******************************idle=1
IF AutoFlow=0 AND NOT(NOT(SystemReadyStatus) OR ErrorState OR Error_PB_Estop1 OR Error_PB_Estop2 OR NOT(AutoStatus)) THEN
	AutoFlow:=1;
END_IF;
IF Autoflow=4 AND LS_S7_MoveBack1 AND LS_S7_MoveBack2 AND LS_S7_MoveBack3 AND LS_S7_MoveBack4 THEN
	Autoflow:=1;
END_IF;
//*******************************推出=2
IF AutoFlow=1 AND
	MachineRunStatus AND
	NOT(IndexData7.FinishFlag[7]) THEN
	AutoFlow:=2;
END_IF;
IF Autoflow=2 AND IndexData7.OKFlag_1[6] THEN
	pushFlag1:=TRUE;
END_IF;
IF Autoflow=2 AND IndexData7.OKFlag_2[5] THEN
	pushFlag2:=TRUE;
END_IF;
IF Autoflow=2 AND IndexData7.OKFlag_3[6] THEN
	pushFlag3:=TRUE;
END_IF;
IF Autoflow=2 AND IndexData7.OKFlag_4[5] THEN
	pushFlag4:=TRUE;
END_IF;
//*******************************推到位=3
IF AutoFlow=2 AND
	(LS_S7_MoveOut1 OR NOT(pushFlag1)) AND
	(LS_S7_MoveOut2 OR NOT(pushFlag2)) AND
	(LS_S7_MoveOut3 OR NOT(pushFlag3)) AND
	(LS_S7_MoveOut4 OR NOT(pushFlag4))
	THEN
	AutoFlow:=3;
END_IF;
RTRIG1(Clk:=pushFlag1);
RTRIG2(Clk:=pushFlag2);
RTRIG3(Clk:=pushFlag3);
RTRIG4(Clk:=pushFlag4);
IF RTRIG1.Q THEN
	OKCount:=OKCount+1;
	TotalCount:=TotalCount+1;
END_IF;
IF RTRIG2.Q THEN
	OKCount:=OKCount+1;
	TotalCount:=TotalCount+1;
END_IF;
IF RTRIG3.Q THEN
	OKCount:=OKCount+1;
	TotalCount:=TotalCount+1;
END_IF;
IF RTRIG4.Q THEN
	OKCount:=OKCount+1;
	TotalCount:=TotalCount+1;
END_IF;
IF pushFlag1 AND LS_S7_MoveOut1 THEN
	IndexData7.OKFlag_1[7]:=TRUE;
	pushFlag1:=FALSE;
END_IF;
IF pushFlag2 AND LS_S7_MoveOut2 THEN
	IndexData7.OKFlag_2[7]:=TRUE;
	pushFlag2:=FALSE;
END_IF;
IF pushFlag3 AND LS_S7_MoveOut3 THEN
	IndexData7.OKFlag_3[7]:=TRUE;
	pushFlag3:=FALSE;
END_IF;
IF pushFlag4 AND LS_S7_MoveOut4 THEN
	IndexData7.OKFlag_4[7]:=TRUE;
	pushFlag4:=FALSE;
END_IF;
//*******************************推回=4
TON1(In:=Autoflow=3, PT:=t#1s);
IF AutoFlow=3 AND TON1.Q	THEN
	AutoFlow:=4;
END_IF;
END_PROGRAM

PROGRAM prStation8
VAR
    SolMove : fbSingleSolRy;
    ErrorState : BOOL;
    AutoFlow : INT;
    TON2 : TON;
END_VAR
VAR_EXTERNAL
    HMIPB_SOL_S8_Move : BOOL;
    AutoStatus : bool;
    SNR_Index : BOOL;
    RY_Index : BOOL;
    SOL_S8_Move : BOOL;
    Error_PB_Estop1 : BOOL;
    Error_PB_Estop2 : BOOL;
    IndexData8 : StationRecord;
    Error_LS_S8_MoveBack : BOOL;
    Error_LS_S8_MoveOut : BOOL;
    SystemReadyStatus : bool;
    MachineRunStatus : bool;
    LS_S8_MoveOut : BOOL;
    LS_S8_MoveBack : BOOL;
END_VAR
SolMove(
	inPushButton:=HMIPB_SOL_S8_Move,
	inAutoStatus:=AutoStatus,
	inAutoFlowSet:=AutoFlow=2,
	inAutoFlowReset:=AutoFlow=3 OR ErrorState,
	inInterLockBack:=TRUE,
	inInterLockOut:=SNR_Index AND NOT(RY_Index),
	outSol=>SOL_S8_Move);
(*************************************************************************************************************)
(*本站狀態判斷*)
IF (IndexData8.OKFlag_1[8]) AND
	(IndexData8.OKFlag_2[8]) AND
	(IndexData8.OKFlag_3[8]) AND
	(IndexData8.OKFlag_4[8])
THEN
	IndexData8.FinishFlag[8]:=TRUE;
END_IF;
(*異常*)
ErrorState:=
Error_LS_S8_MoveBack OR
Error_LS_S8_MoveOut;
//*********************************自動********************************************
//****************************power on=0
IF NOT(SystemReadyStatus) OR ErrorState OR Error_PB_Estop1 OR Error_PB_Estop2 THEN
	Autoflow:=0;
END_IF;
//*******************************idle=1
IF AutoFlow=0 AND NOT(NOT(SystemReadyStatus) OR ErrorState OR Error_PB_Estop1 OR Error_PB_Estop2 ) THEN
	AutoFlow:=1;
END_IF;
IF AutoFlow=3 AND LS_S8_MoveBack THEN
	AutoFlow:=1;
END_IF;
//*******************************推出=2
IF AutoFlow=1 AND
	NOT(IndexData8.FinishFlag[8]) THEN
	AutoFlow:=2;
END_IF;

TON2(In:=AutoFlow=2 AND LS_S8_MoveOut, PT:=t#1s);
//*******************************推回=3
IF AutoFlow=2 AND TON2.Q THEN
	AutoFlow:=3;
	
	IndexData8.OKFlag_1[8]:=TRUE;
	IndexData8.OKFlag_2[8]:=TRUE;
	IndexData8.OKFlag_3[8]:=TRUE;
	IndexData8.OKFlag_4[8]:=TRUE;
END_IF;
END_PROGRAM

PROGRAM prStart
VAR
    R_TRIG1 : R_TRIG;
END_VAR
VAR_EXTERNAL
    PB_Start1 : BOOL;
    PB_Start2 : BOOL;
    PB_Estop1 : BOOL;
    PB_Estop2 : BOOL;
    PB_Reset1 : BOOL;
    MachineRunStatus : bool;
    PB_Reset2 : BOOL;
    ErrorStatus_MachineStop : bool;
    AutoStatus : bool;
END_VAR
//start
R_TRIG1(Clk:=PB_Start1 OR PB_Start2);
IF R_TRIG1.Q AND (PB_Estop1) AND (PB_Estop2) AND NOT(ErrorStatus_MachineStop) AND AutoStatus THEN
	MachineRunStatus:=TRUE;
END_IF;
//stop
IF PB_Reset1 OR PB_Reset2 OR NOT(PB_Estop1) OR NOT(PB_Estop2) OR ErrorStatus_MachineStop THEN
	MachineRunStatus:=FALSE;
END_IF;
END_PROGRAM

PROGRAM prError
VAR
    ErrorS2Move : fbErrorSOL_S;
    ErrorS2TH1 : fbErrorSOL_D;
    ErrorS2TH2 : fbErrorSOL_D;
    ErrorS3Move : fbErrorSOL_S;
    ErrorS3TH1 : fbErrorSOL_D;
    ErrorS3TH2 : fbErrorSOL_D;
    ErrorS5Fix : fbErrorSOL_S;
    ErrorS5UpDown : fbErrorSOL_S;
    ErrorS6Fix : fbErrorSOL_S;
    ErrorS6UpDown : fbErrorSOL_S;
    ErrorS7Move1 : fbErrorSOL_S;
    ErrorS7Move2 : fbErrorSOL_S;
    ErrorS7Move3 : fbErrorSOL_S;
    ErrorS7Move4 : fbErrorSOL_S;
    ErrorS8Move : fbErrorSOL_S;
    TON1 : TON;
    TON2 : TON;
    ErrorS5Index : fbErrorSOL_D;
    ErrorS6Index : fbErrorSOL_D;
END_VAR
VAR_EXTERNAL
    AutoStatus : bool;
    PB_Reset1 : BOOL;
    PB_Reset2 : BOOL;
    SOL_S2_Move : BOOL;
    LS_S2_MoveBack : BOOL;
    LS_S2_MoveOut : BOOL;
    Error_LS_S2_MoveBack : BOOL;
    Error_LS_S2_MoveOut : BOOL;
    SOL_S2_THBack1 : BOOL;
    SOL_S2_THOut1 : BOOL;
    LS_S2_THBack1 : BOOL;
    LS_S2_THOut1 : BOOL;
    Error_LS_S2_THBack1 : BOOL;
    Error_LS_S2_THOut1 : BOOL;
    SOL_S2_THBack2 : BOOL;
    SOL_S2_THOut2 : BOOL;
    LS_S2_THBack2 : BOOL;
    LS_S2_THOut2 : BOOL;
    Error_LS_S2_THBack2 : BOOL;
    Error_LS_S2_THOut2 : BOOL;
    SOL_S3_Move : BOOL;
    LS_S3_MoveBack : BOOL;
    LS_S3_MoveOut : BOOL;
    Error_LS_S3_MoveBack : BOOL;
    Error_LS_S3_MoveOut : BOOL;
    SOL_S3_THBack1 : BOOL;
    SOL_S3_THOut1 : BOOL;
    LS_S3_THBack1 : BOOL;
    LS_S3_THOut1 : BOOL;
    Error_LS_S3_THBack1 : BOOL;
    Error_LS_S3_THOut1 : BOOL;
    SOL_S3_THBack2 : BOOL;
    SOL_S3_THOut2 : BOOL;
    LS_S3_THBack2 : BOOL;
    LS_S3_THOut2 : BOOL;
    Error_LS_S3_THBack2 : BOOL;
    Error_LS_S3_THOut2 : BOOL;
    SOL_S5_Fix : BOOL;
    LS_S5_FixBack : BOOL;
    LS_S5_FixOut : BOOL;
    Error_LS_S5_FixBack : BOOL;
    Error_LS_S5_FixOut : BOOL;
    SOL_S5_UpDown : BOOL;
    LS_S5_UpDownBack : BOOL;
    LS_S5_UpDownOut : BOOL;
    Error_LS_S5_UpDownBack : BOOL;
    Error_LS_S5_UpDownOut : BOOL;
    SOL_S6_Fix : BOOL;
    LS_S6_FixBack : BOOL;
    LS_S6_FixOut : BOOL;
    Error_LS_S6_FixBack : BOOL;
    Error_LS_S6_FixOut : BOOL;
    SOL_S6_UpDown : BOOL;
    LS_S6_UpDownBack : BOOL;
    LS_S6_UpDownOut : BOOL;
    Error_LS_S6_UpDownBack : BOOL;
    Error_LS_S6_UpDownOut : BOOL;
    SOL_S7_Move1 : BOOL;
    LS_S7_MoveBack1 : BOOL;
    LS_S7_MoveOut1 : BOOL;
    Error_LS_S7_MoveBack1 : BOOL;
    Error_LS_S7_MoveOut1 : BOOL;
    SOL_S7_Move2 : BOOL;
    LS_S7_MoveBack2 : BOOL;
    LS_S7_MoveOut2 : BOOL;
    Error_LS_S7_MoveBack2 : BOOL;
    Error_LS_S7_MoveOut2 : BOOL;
    SOL_S7_Move3 : BOOL;
    LS_S7_MoveBack3 : BOOL;
    LS_S7_MoveOut3 : BOOL;
    Error_LS_S7_MoveBack3 : BOOL;
    Error_LS_S7_MoveOut3 : BOOL;
    SOL_S7_Move4 : BOOL;
    LS_S7_MoveBack4 : BOOL;
    LS_S7_MoveOut4 : BOOL;
    Error_LS_S7_MoveBack4 : BOOL;
    Error_LS_S7_MoveOut4 : BOOL;
    SOL_S8_Move : BOOL;
    LS_S8_MoveBack : BOOL;
    LS_S8_MoveOut : BOOL;
    Error_LS_S8_MoveBack : BOOL;
    Error_LS_S8_MoveOut : BOOL;
    RY_Index : BOOL;
    Error_SNR_Index : BOOL;
    SOL_S5_IndexFixBack : BOOL;
    SOL_S5_IndexFixOut : BOOL;
    LS_S5_IndexFixBack : BOOL;
    LS_S5_IndexFixOut : BOOL;
    Error_LS_S5_IndexFixBack : BOOL;
    Error_LS_S5_IndexFixOut : BOOL;
    Error_LS_S6_IndexFixOut : BOOL;
    Error_LS_S6_IndexFixBack : BOOL;
    LS_S6_IndexFixOut : BOOL;
    LS_S6_IndexFixBack : BOOL;
    SOL_S6_IndexFixOut : BOOL;
    SOL_S6_IndexFixBack : BOOL;
    ErrorStatus_MachineStop : bool;
    Error_SNR_AirSource : BOOL;
    Error_SNR_S2_Feed : BOOL;
    Error_SNR_S3_Feed : BOOL;
    Error_SNR_S5_L_Feed : BOOL;
    Error_SNR_S5_R_Feed : BOOL;
    Error_SNR_S6_L_Feed : BOOL;
    Error_SNR_S6_R_Feed : BOOL;
    Error_SNR_S7_Full : BOOL;
    SNR_AirSource : BOOL;
    MachineRunStatus : bool;
    SNR_S7_Full : BOOL;
    ErrorStatus_MachineNonStop : bool;
    Error_SNR_S2_Full : BOOL;
    Error_SNR_S3_Full : BOOL;
    Error_SNR_S5_Full : BOOL;
    Error_SNR_S6_Full : BOOL;
END_VAR
//**********************************************************s2
ErrorS2Move(
	bAutoStatus:=AutoStatus,
	bResetPB:=PB_Reset1 OR PB_Reset2,
	bSOL:=SOL_S2_Move,
	bBackLS:=LS_S2_MoveBack,
	bOutLS:=LS_S2_MoveOut,
	bErrorStatus_Back=>Error_LS_S2_MoveBack,
	bErrorStatus_Out=>Error_LS_S2_MoveOut);
ErrorS2TH1(
	bAutoStatus:=AutoStatus,
	bResetPB:=PB_Reset1 OR PB_Reset2,
	bBackSOL:=SOL_S2_THBack1,
	bOutSOL:=SOL_S2_THOut1,
	bBackLS:=LS_S2_THBack1,
	bOutLS:=LS_S2_THOut1,
	bErrorStatus_Back=>Error_LS_S2_THBack1,
	bErrorStatus_Out=>Error_LS_S2_THOut1);
ErrorS2TH2(
	bAutoStatus:=AutoStatus,
	bResetPB:=PB_Reset1 OR PB_Reset2,
	bBackSOL:=SOL_S2_THBack2,
	bOutSOL:=SOL_S2_THOut2,
	bBackLS:=LS_S2_THBack2,
	bOutLS:=LS_S2_THOut2,
	bErrorStatus_Back=>Error_LS_S2_THBack2,
	bErrorStatus_Out=>Error_LS_S2_THOut2);
//**********************************************************s3
ErrorS3Move(
	bAutoStatus:=AutoStatus,
	bResetPB:=PB_Reset1 OR PB_Reset2,
	bSOL:=SOL_S3_Move,
	bBackLS:=LS_S3_MoveBack,
	bOutLS:=LS_S3_MoveOut,
	bErrorStatus_Back=>Error_LS_S3_MoveBack,
	bErrorStatus_Out=>Error_LS_S3_MoveOut);
ErrorS3TH1(
	bAutoStatus:=AutoStatus,
	bResetPB:=PB_Reset1 OR PB_Reset2,
	bBackSOL:=SOL_S3_THBack1,
	bOutSOL:=SOL_S3_THOut1,
	bBackLS:=LS_S3_THBack1,
	bOutLS:=LS_S3_THOut1,
	bErrorStatus_Back=>Error_LS_S3_THBack1,
	bErrorStatus_Out=>Error_LS_S3_THOut1);
ErrorS3TH2(
	bAutoStatus:=AutoStatus,
	bResetPB:=PB_Reset1 OR PB_Reset2,
	bBackSOL:=SOL_S3_THBack2,
	bOutSOL:=SOL_S3_THOut2,
	bBackLS:=LS_S3_THBack2,
	bOutLS:=LS_S3_THOut2,
	bErrorStatus_Back=>Error_LS_S3_THBack2,
	bErrorStatus_Out=>Error_LS_S3_THOut2);
//**********************************************************s5
ErrorS5Fix(
	bAutoStatus:=AutoStatus,
	bResetPB:=PB_Reset1 OR PB_Reset2,
	bSOL:=SOL_S5_Fix,
	bBackLS:=LS_S5_FixBack,
	bOutLS:=LS_S5_FixOut,
	bErrorStatus_Back=>Error_LS_S5_FixBack,
	bErrorStatus_Out=>Error_LS_S5_FixOut);
ErrorS5UpDown(
	bAutoStatus:=AutoStatus,
	bResetPB:=PB_Reset1 OR PB_Reset2,
	bSOL:=SOL_S5_UpDown,
	bBackLS:=LS_S5_UpDownBack,
	bOutLS:=LS_S5_UpDownOut,
	bErrorStatus_Back=>Error_LS_S5_UpDownBack,
	bErrorStatus_Out=>Error_LS_S5_UpDownOut);
//**********************************************************s6
ErrorS6Fix(
	bAutoStatus:=AutoStatus,
	bResetPB:=PB_Reset1 OR PB_Reset2,
	bSOL:=SOL_S6_Fix,
	bBackLS:=LS_S6_FixBack,
	bOutLS:=LS_S6_FixOut,
	bErrorStatus_Back=>Error_LS_S6_FixBack,
	bErrorStatus_Out=>Error_LS_S6_FixOut);
ErrorS6UpDown(
	bAutoStatus:=AutoStatus,
	bResetPB:=PB_Reset1 OR PB_Reset2,
	bSOL:=SOL_S6_UpDown,
	bBackLS:=LS_S6_UpDownBack,
	bOutLS:=LS_S6_UpDownOut,
	bErrorStatus_Back=>Error_LS_S6_UpDownBack,
	bErrorStatus_Out=>Error_LS_S6_UpDownOut);
//**********************************************************s7
ErrorS7Move1(
	bAutoStatus:=AutoStatus,
	bResetPB:=PB_Reset1 OR PB_Reset2,
	bSOL:=SOL_S7_Move1,
	bBackLS:=LS_S7_MoveBack1,
	bOutLS:=LS_S7_MoveOut1,
	bErrorStatus_Back=>Error_LS_S7_MoveBack1,
	bErrorStatus_Out=>Error_LS_S7_MoveOut1);
ErrorS7Move2(
	bAutoStatus:=AutoStatus,
	bResetPB:=PB_Reset1 OR PB_Reset2,
	bSOL:=SOL_S7_Move2,
	bBackLS:=LS_S7_MoveBack2,
	bOutLS:=LS_S7_MoveOut2,
	bErrorStatus_Back=>Error_LS_S7_MoveBack2,
	bErrorStatus_Out=>Error_LS_S7_MoveOut2);
ErrorS7Move3(
	bAutoStatus:=AutoStatus,
	bResetPB:=PB_Reset1 OR PB_Reset2,
	bSOL:=SOL_S7_Move3,
	bBackLS:=LS_S7_MoveBack3,
	bOutLS:=LS_S7_MoveOut3,
	bErrorStatus_Back=>Error_LS_S7_MoveBack3,
	bErrorStatus_Out=>Error_LS_S7_MoveOut3);
ErrorS7Move4(
	bAutoStatus:=AutoStatus,
	bResetPB:=PB_Reset1 OR PB_Reset2,
	bSOL:=SOL_S7_Move4,
	bBackLS:=LS_S7_MoveBack4,
	bOutLS:=LS_S7_MoveOut4,
	bErrorStatus_Back=>Error_LS_S7_MoveBack4,
	bErrorStatus_Out=>Error_LS_S7_MoveOut4);
//**********************************************************s8
ErrorS8Move(
	bAutoStatus:=AutoStatus,
	bResetPB:=PB_Reset1 OR PB_Reset2,
	bSOL:=SOL_S8_Move,
	bBackLS:=LS_S8_MoveBack,
	bOutLS:=LS_S8_MoveOut,
	bErrorStatus_Back=>Error_LS_S8_MoveBack,
	bErrorStatus_Out=>Error_LS_S8_MoveOut);
//**********************************************************轉盤微動開關
TON1(IN:= RY_Index ,PT:= t#6s);
IF TON1.Q THEN
	Error_SNR_Index:=TRUE;
END_IF;
ErrorS5Index(
	bAutoStatus:=AutoStatus,
	bResetPB:=PB_Reset1 OR PB_Reset2,
	bBackSOL:=SOL_S5_IndexFixBack,
	bOutSOL:=SOL_S5_IndexFixOut,
	bBackLS:=LS_S5_IndexFixBack,
	bOutLS:=LS_S5_IndexFixOut,
	bErrorStatus_Back=>Error_LS_S5_IndexFixBack,
	bErrorStatus_Out=>Error_LS_S5_IndexFixOut);
ErrorS6Index(
	bAutoStatus:=AutoStatus,
	bResetPB:=PB_Reset1 OR PB_Reset2,
	bBackSOL:=SOL_S6_IndexFixBack,
	bOutSOL:=SOL_S6_IndexFixOut,
	bBackLS:=LS_S6_IndexFixBack,
	bOutLS:=LS_S6_IndexFixOut,
	bErrorStatus_Back=>Error_LS_S6_IndexFixBack,
	bErrorStatus_Out=>Error_LS_S6_IndexFixOut);
//**********************************************************氣源
IF MachineRunStatus AND NOT(SNR_AirSource) THEN
	Error_SNR_AirSource:=TRUE;
END_IF;
IF PB_Reset1 OR PB_Reset2 THEN
	Error_SNR_AirSource:=FALSE;
END_IF;
//**********************************************************ST7滿料
TON2(In:=SNR_S7_Full,PT:=t#3s);
IF TON2.Q THEN
	Error_SNR_S7_Full:=TRUE;
END_IF;
IF PB_Reset1 OR PB_Reset2 THEN
	Error_SNR_S7_Full:=FALSE;
END_IF;
//**********************************************************
ErrorStatus_MachineNonStop:=
Error_SNR_S2_Full OR
Error_SNR_S3_Full OR
Error_SNR_S5_Full OR
Error_SNR_S6_Full;
//**********************************************************
ErrorStatus_MachineStop:=
Error_LS_S2_MoveBack OR
Error_LS_S2_MoveOut OR
Error_LS_S2_THBack1 OR 
Error_LS_S2_THBack2 OR
Error_LS_S2_THOut1 OR
Error_LS_S2_THOut2 OR
Error_LS_S3_MoveBack OR
Error_LS_S3_MoveOut OR
Error_LS_S3_THBack1 OR
Error_LS_S3_THBack2 OR
Error_LS_S3_THOut1 OR
Error_LS_S3_THOut2 OR
Error_LS_S5_FixBack OR
Error_LS_S5_FixOut OR
Error_LS_S5_IndexFixBack OR 
Error_LS_S5_IndexFixOut OR
Error_LS_S5_UpDownBack OR
Error_LS_S5_UpDownOut OR
Error_LS_S6_FixBack OR
Error_LS_S6_FixOut OR
Error_LS_S6_IndexFixBack OR 
Error_LS_S6_IndexFixOut OR
Error_LS_S6_UpDownBack OR
Error_LS_S6_UpDownOut OR
Error_LS_S7_MoveBack1 or
Error_LS_S7_MoveBack2 or
Error_LS_S7_MoveBack3 or
Error_LS_S7_MoveBack4 or
Error_LS_S7_MoveOut1 or
Error_LS_S7_MoveOut2 or
Error_LS_S7_MoveOut3 or
Error_LS_S7_MoveOut4 or
Error_LS_S8_MoveBack OR
Error_LS_S8_MoveOut OR
Error_SNR_AirSource OR
Error_SNR_Index OR
Error_SNR_S2_Feed OR
Error_SNR_S3_Feed OR
Error_SNR_S5_L_Feed OR
Error_SNR_S5_R_Feed OR
Error_SNR_S6_L_Feed OR
Error_SNR_S6_R_Feed OR
Error_SNR_S7_Full;
END_PROGRAM

PROGRAM prCommProgram
VAR
    statusFlash1s : BOOL;
    bClock : BOOL;
    TON1 : TON;
    TON2 : TON;
    R_TRIG1 : R_TRIG;
END_VAR
VAR_EXTERNAL
    Flash1s : BOOL;
    HMIPB_ResetCount : BOOL;
    HMI_AllCount : UDINT;
END_VAR
//bClock:=Get1sClk();
IF HMIPB_ResetCount THEN
	HMI_AllCount:=0;
END_IF;
//flsash 1s
TON1(In:=NOT(statusFlash1s), PT:=t#1s);
TON2(In:=(statusFlash1s), PT:=t#1s);
IF TON1.Q THEN
	bClock:=TRUE;
END_IF;
IF TON2.Q THEN
	bClock:=FALSE;
END_IF;
Flash1s:=bClock;
statusFlash1s:=Flash1s;
END_PROGRAM

PROGRAM prBZAndLight
VAR_EXTERNAL
    Flash1s : BOOL;
    GL : BOOL;
    YL : BOOL;
    SystemReadyStatus : bool;
    ErrorStatus_MachineNonStop : bool;
    ErrorStatus_MachineStop : bool;
    RL : BOOL;
    BZ : BOOL;
    MachineRunStatus : bool;
END_VAR
(*BZ*)	
IF (ErrorStatus_MachineStop OR ErrorStatus_MachineNonStop) THEN
	BZ:=Flash1s;
	ELSE
	BZ:=FALSE;
END_IF;
//(*紅燈長亮:異常*)
IF SystemReadyStatus AND (ErrorStatus_MachineStop) THEN
	RL:=TRUE;
	ELSE
	RL:=FALSE;
END_IF;
(*綠燈閃爍:運轉,長亮:待機*)
IF SystemReadyStatus AND NOT(ErrorStatus_MachineNonStop) AND NOT(ErrorStatus_MachineStop)  THEN
	IF MachineRunStatus THEN
		GL:=Flash1s;
	ELSE
		GL:=TRUE;
	END_IF;
	ELSE
	GL:=FALSE;
END_IF;
(*黃燈閃爍:振動筒缺料*)
IF SystemReadyStatus AND ErrorStatus_MachineNonStop AND NOT(ErrorStatus_MachineStop) THEN
	YL:=Flash1s;
	ELSE
	YL:=FALSE;
END_IF;
END_PROGRAM

PROGRAM prCycleTime
VAR
    TON1 : TON;
    tCycleTime : TIME;
    RTRIG1 : R_TRIG;
    cycle : LINT;
    FTRIG1 : F_TRIG;
END_VAR
VAR_EXTERNAL
    HMI_CycleTime : LINT;
    MachineRunStatus : bool;
    SNR_Index : BOOL;
END_VAR
IF FTRIG1.Q THEN
	HMI_CycleTime:=cycle;
END_IF;
TON1(In:=MachineRunStatus AND SNR_Index, PT:=t#1m,ET=>tCycleTime);
IF MachineRunStatus AND SNR_Index THEN
	cycle:=TimeToNanoSec(tCycleTime)/10000000;
END_IF;
FTRIG1(Clk:=SNR_Index);
END_PROGRAM

PROGRAM prStation5
VAR
    SolFix : fbSingleSolRy;
    SolUpDown : fbSingleSolRy;
    SolClamp : fbSingleSolRy;
    ErrorState : BOOL;
    TON1 : TON;
    TON2 : TON;
    oldTorqueR : LREAL;
    screwR : UINT;
    oldTorqueL : LREAL;
    screwL : UINT;
    AutoFlow : INT;
    ScrewLeft : fbScrewFlow;
    ScrewRight : fbScrewFlow;
    TON3 : TON;
END_VAR
VAR_EXTERNAL
    HMIPB_SOL_S5_Fix : BOOL;
    AutoStatus : bool;
    SNR_Index : BOOL;
    RY_Index : BOOL;
    SOL_S5_Fix : BOOL;
    HMIPB_SOL_S5_UpDown : BOOL;
    SOL_S5_UpDown : BOOL;
    HMIPB_SOL_S5_Clamp : BOOL;
    SOL_S5_Clamp : BOOL;
    Error_PB_Estop1 : BOOL;
    Error_PB_Estop2 : BOOL;
    IndexData5 : StationRecord;
    Error_LS_S5_FixBack : BOOL;
    Error_LS_S5_FixOut : BOOL;
    Error_LS_S5_UpDownBack : BOOL;
    Error_LS_S5_UpDownOut : BOOL;
    LS_S5_UpDownOut : BOOL;
    LS_S5_UpDownBack : BOOL;
    SystemReadyStatus : bool;
    LS_S5_FixBack : BOOL;
    MachineRunStatus : bool;
    ScrewStartFlag : ARRAY[0..3] OF bool;
    SNR_S5_R_Check : BOOL;
    HMIPB_FW_AxisRSt5 : BOOL;
    HMI_ScrewTorque_St5_R : LREAL;
    HMIPB_RW_AxisRSt5 : BOOL;
    SNR_S5_L_Check : BOOL;
    HMIPB_FW_AxisLSt5 : BOOL;
    HMI_ScrewTorque_St5_L : LREAL;
    HMIPB_RW_AxisLSt5 : BOOL;
    HMIShow_CurrentSpeed : ARRAY[0..3] OF LREAL;
    FeedStartFlag : ARRAY[0..1] OF bool;
    OBJScrewInClip : ARRAY[0..3] OF INT;
    Error_SNR_S5_L_Feed : BOOL;
    Error_SNR_S5_R_Feed : BOOL;
END_VAR
VAR_EXTERNAL CONSTANT
    MC_AxisLSt5 : _sAXIS_REF;
END_VAR
VAR_EXTERNAL
    ScrewStartS5LFW : BOOL;
    ScrewStartS5LRW : BOOL;
END_VAR
VAR_EXTERNAL CONSTANT
    MC_AxisRSt5 : _sAXIS_REF;
END_VAR
VAR_EXTERNAL
    HMIShow_CurrentTorque : ARRAY[0..3] OF LREAL;
    ScrewStartS5RFW : BOOL;
    ScrewStartS5RRW : BOOL;
    HMI_BackOutTorque_St5_L : LREAL;
    HMI_BackOutTorque_St5_R : LREAL;
    SOL_S5_Feed : BOOL;
    HMIShow_CurrentPosition : ARRAY[0..3] OF LREAL;
    HMI_LimitAngle_St5_L : LREAL;
    HMI_LimitAngle_St5_R : LREAL;
    ResetAddress : ARRAY[0..3] OF bool;
    HMI_BackOutAngle_St5_L : LREAL;
    HMI_ScrewSpeed_St5_L : LREAL;
    HMI_BackOutAngle_St5_R : LREAL;
    HMI_ScrewSpeed_St5_R : LREAL;
    BackoutBusy : ARRAY[0..3] OF BOOL;
    BackoutStart : ARRAY[0..3] OF BOOL;
    HMI_NoScrewAngle_St5_L : LREAL;
    HMI_NoScrewAngle_St5_R : LREAL;
    HMI_Find_St5_L : LINT;
    HMI_Find_St5_R : LINT;
END_VAR
SolFix(
	inPushButton:=HMIPB_SOL_S5_Fix,
	inAutoStatus:=AutoStatus,
	inAutoFlowSet:=Autoflow=2,
	inAutoFlowReset:=Autoflow=4 OR ErrorState,
	inInterLockBack:=TRUE,
	inInterLockOut:=SNR_Index AND NOT(RY_Index),
	outSol=>SOL_S5_Fix);
SolUpDown(
	inPushButton:=HMIPB_SOL_S5_UpDown,
	inAutoStatus:=AutoStatus,
	inAutoFlowSet:=AutoFlow=2,
	inAutoFlowReset:=Autoflow=4 OR ErrorState,
	inInterLockBack:=TRUE,
	inInterLockOut:=SNR_Index AND NOT(RY_Index),
	outSol=>SOL_S5_UpDown);
SolClamp(
	inPushButton:=HMIPB_SOL_S5_Clamp,
	inAutoStatus:=AutoStatus,
	inAutoFlowSet:=SOL_S5_UpDown AND LS_S5_UpDownOut AND AutoStatus AND (screwR>=2 AND screwR<20 AND screwL>=2 AND screwL<20),
	inAutoFlowReset:=(LS_S5_UpDownBack AND NOT(SOL_S5_UpDown) AND AutoStatus) OR ErrorState,
	inInterLockBack:=TRUE,
	inInterLockOut:=TRUE,
	outSol=>SOL_S5_Clamp);
TON3(In:=SOL_S5_UpDown AND LS_S5_UpDownOut AND AutoStatus,PT:=t#500ms);
(*************************************************************************************************************)
(*EStOP and Error*)
IF (Error_PB_Estop1 OR Error_PB_Estop2) AND NOT(IndexData5.OKFlag_4[5]) THEN
	IndexData5.NGFlag_4[5]:=TRUE;
	IndexData5.ErrorRecordData[5]:=1;
END_IF;
IF (Error_PB_Estop1 OR Error_PB_Estop2) AND NOT(IndexData5.OKFlag_2[5]) THEN
	IndexData5.NGFlag_2[5]:=TRUE;
	IndexData5.ErrorRecordData[5]:=1;
END_IF;
IF ErrorState AND NOT(IndexData5.OKFlag_4[5]) THEN
	IndexData5.NGFlag_4[5]:=TRUE;
	IndexData5.ErrorRecordData[5]:=2;
END_IF;
IF ErrorState AND NOT(IndexData5.OKFlag_2[5]) THEN
	IndexData5.NGFlag_2[5]:=TRUE;
	IndexData5.ErrorRecordData[5]:=2;
END_IF;
(*本站狀態判斷*)
IF (IndexData5.OKFlag_4[5] OR IndexData5.NGFlag_4[5]) AND
	(IndexData5.OKFlag_2[5] OR IndexData5.NGFlag_2[5])
	THEN
	IndexData5.FinishFlag[5]:=TRUE;
END_IF;
(*前站判斷*)
IF IndexData5.NGFlag_4[2] OR NOT(IndexData5.OKFlag_4[2]) THEN
	IndexData5.NGFlag_4[5]:=TRUE;
END_IF;
IF IndexData5.NGFlag_2[2] OR NOT(IndexData5.OKFlag_2[2]) THEN
	IndexData5.NGFlag_2[5]:=TRUE;
END_IF;
(*異常*)
ErrorState:=
Error_LS_S5_FixBack OR
Error_LS_S5_FixOut OR
Error_LS_S5_UpDownBack OR
Error_LS_S5_UpDownOut;
//無螺絲

//*********************************自動********************************************
//****************************power on=0
IF NOT(SystemReadyStatus) OR ErrorState OR Error_PB_Estop1 OR Error_PB_Estop2 OR NOT(AutoStatus) THEN
	Autoflow:=0;
END_IF;
//****************************idle=1
IF AutoFlow=0 AND NOT(NOT(SystemReadyStatus) OR ErrorState OR Error_PB_Estop1 OR Error_PB_Estop2 OR NOT(AutoStatus)) THEN
	AutoFlow:=1;
END_IF;
IF Autoflow=4 AND screwL=1 AND screwR=1 AND LS_S5_FixBack AND LS_S5_UpDownBack THEN
	SOL_S5_Clamp:=FALSE;
	Autoflow:=1;
END_IF;
//****************************定位出,向下,鎖付開始=2
IF AutoFlow=1 AND
	NOT(FeedStartFlag[0]) AND
	NOT(Error_SNR_S5_L_Feed) AND
	NOT(Error_SNR_S5_R_Feed) AND
	NOT(SOL_S5_Feed) AND
	SNR_Index AND
	NOT(RY_Index) AND
	MachineRunStatus AND
	NOT(IndexData5.FinishFlag[5]) THEN
	ScrewStartFlag[0]:=TRUE;
	ScrewStartFlag[1]:=TRUE;
	Autoflow:=2;
END_IF;
//****************************鎖付OK=3
IF Autoflow=2 AND screwL=8 THEN//鎖付OK
	ScrewStartFlag[0]:=FALSE;
	IndexData5.OKFlag_4[5]:=TRUE;
END_IF;
IF Autoflow=2 AND screwL=9999 THEN//鎖付NG
	ScrewStartFlag[0]:=FALSE;
	IndexData5.NGFlag_4[5]:=TRUE;
END_IF;
IF Autoflow=2 AND screwR=8 THEN//鎖付OK
	ScrewStartFlag[1]:=FALSE;
	IndexData5.OKFlag_2[5]:=TRUE;
END_IF;
IF Autoflow=2 AND screwR=9999 THEN//鎖付NG
	ScrewStartFlag[1]:=FALSE;
	IndexData5.NGFlag_2[5]:=TRUE;
END_IF;
IF Autoflow=2 AND IndexData5.FinishFlag[5] THEN
	Autoflow:=3;
END_IF;
//****************************向上,定位回=4
IF Autoflow=3 AND LS_S5_UpDownOut AND NOT(ScrewStartFlag[0]) AND NOT(ScrewStartFlag[1]) THEN
	Autoflow:=4;
END_IF;
IF LS_S5_UpDownOut AND SOL_S5_UpDown AND AutoStatus THEN
	FeedStartFlag[0]:=TRUE;
END_IF;
ScrewLeft(
	inStartFlag:=ScrewStartFlag[0],
	inCheckSensor:=SNR_S5_L_Check,
	inStopFlag:= MC_AxisLSt5.Status.Standstill,
	inBackoutBusy:=BackoutBusy[0],
	inCMDTorque:=HMI_BackOutTorque_St5_L,
	inCMDAddress:=HMI_LimitAngle_St5_L,
	inNoScrewSetAngle:=HMI_NoScrewAngle_St5_L,
	inFindTime:=HMI_Find_St5_L,
	inTorqueValue:=HMIShow_CurrentTorque[0],
	inAddressValue:=HMIShow_CurrentPosition[0],
	outFW=>ScrewStartS5LFW,
	outRW=>ScrewStartS5LRW,
	outBackout=>BackoutStart[0],
	outFlowNo=> screwL,
	outResetAddress=>ResetAddress[0],
	inoutTorque:= HMI_ScrewTorque_St5_L);
ScrewRight(
	inStartFlag:=ScrewStartFlag[1],
	inCheckSensor:=SNR_S5_R_Check,
	inStopFlag:= MC_AxisRSt5.Status.Standstill,
	inBackoutBusy:=BackoutBusy[1],
	inCMDTorque:=HMI_BackOutTorque_St5_R,
	inCMDAddress:=HMI_LimitAngle_St5_R,
	inNoScrewSetAngle:=HMI_NoScrewAngle_St5_R,
	inFindTime:=HMI_Find_St5_R,
	inTorqueValue:=HMIShow_CurrentTorque[1],
	inAddressValue:=HMIShow_CurrentPosition[1],
	outFW=>ScrewStartS5RFW,
	outRW=>ScrewStartS5RRW,
	outBackout=>BackoutStart[1],
	outFlowNo=> screwR,
	outResetAddress=>ResetAddress[1],
	inoutTorque:= HMI_ScrewTorque_St5_R);
END_PROGRAM

